(* Logix 5000 project; controller STAT 1756-L72 rev 20.12; software revision 20.04; part 2 of 34 *)
(* tags used below, declared in another part *)
   N7 : DINT[255];
   p15 : BOOL;
   P16 : BOOL;
   P17 : BOOL;
   P18 : BOOL;
   P23 : BOOL;
   P24 : BOOL;
   P3 : BOOL;
   P4 : BOOL;
   pd3 : BOOL;
   pd4 : BOOL;
   pd5 : BOOL;
   pd6 : BOOL;
   PD7 : BOOL;
   PD8 : BOOL;
   PM1 : BOOL;
   PM2 : BOOL;
   PM3 : BOOL;
   PM4 : BOOL;
   Q2 : REAL;
   Q3 : REAL;
   Q4 : REAL;
   real : REAL;
   S : INT[164];
   S1 : BOOL;
   Seconde : BOOL;

ADD_ON_INSTRUCTION integrat   (* revision 1.0 *)
VAR_INPUT
   rate : DINT; {required}
END_VAR
VAR_OUTPUT
   oai : DINT; {access Read Only, required}
END_VAR
VAR_INPUT
   AI : DINT; {required}
END_VAR
VAR
   memo : REAL; {access None}
   memo1 : REAL; {access None}
   rate1 : DINT; {access None}
   memo2 : REAL; {access None}
END_VAR

ROUTINE Logic   (* ladder *)
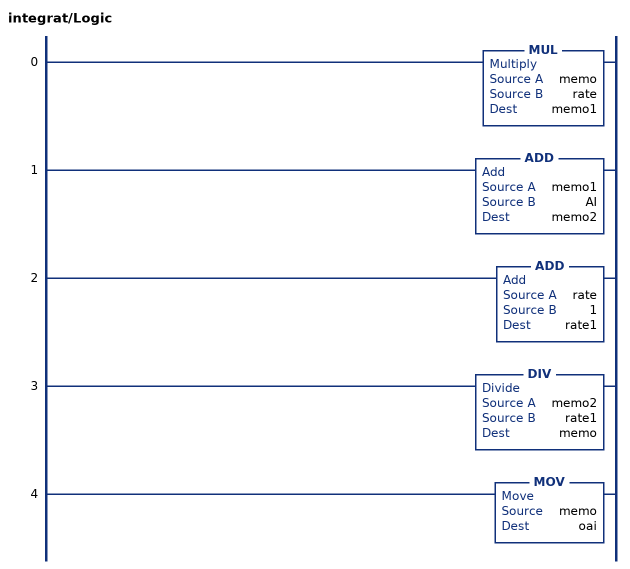
   0: MUL(memo,rate,memo1);
   1: ADD(memo1,AI,memo2);
   2: ADD(rate,1,rate1);
   3: DIV(memo2,rate1,memo);
   4: MOV(memo,oai);
END_ROUTINE
END_ADD_ON_INSTRUCTION

ADD_ON_INSTRUCTION SCP   (* revision 1.2, vendor Rockwell Automation *)
VAR_INPUT
   Input : REAL; {required}
   Input_Min : REAL; {required}
   Input_Max : REAL; {required}
   Scaled_Min : REAL; {required}
   Scaled_Max : REAL; {required}
END_VAR
VAR_OUTPUT
   Output : REAL; {access Read Only, required}
END_VAR
VAR
   Rate : REAL;
END_VAR

ROUTINE Logic   (* ladder *)
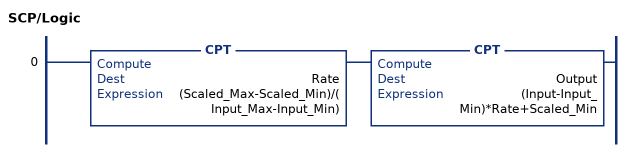
   0: CPT(Rate,(Scaled_Max-Scaled_Min)/(Input_Max-Input_Min))CPT(Output,(Input-Input_Min)*Rate+Scaled_Min);
END_ROUTINE
END_ADD_ON_INSTRUCTION

VAR_GLOBAL   (* controller tags *)
   ai_flow_L1 : REAL := 236.55;
   ai_flow_L2 : REAL := 242.7;
   ai_flow_L3 : REAL := 242.85;
   apport_soude_ibt_occupe : BOOL;
   aux2_P1 : BOOL := 1;
   AUX2_P2 : BOOL := 1;
   AUX_COND_KOELTOREN : REAL := 3777.7964;
   AUX_LVL_KOEL : DINT := 857;
   aux_P1_ETANG : BOOL := 1;
   AUX_P1P2 : BOOL;
   AUX_P2 : BOOL := 1;
   AUX_P5_RINC : BOOL;
   av310 : BOOL := 1;
   av320 : BOOL := 1;
   av330 : BOOL := 1;
   averflowput1 : DINT := -30;
   averflowput2 : DINT := -24;
   averK1 : DINT := 206;
   averK2 : DINT := 230;
   averL1 : DINT := 261;
   averL2 : DINT := 162;
   averL3 : DINT := 242;
   averlpmpput2 : DINT;
   averpmpput1 : DINT;
   averQ1 : DINT := 170;
   averQ2 : DINT := 131;
   B10 : DINT[20] := ([0] := 2#0000_0000_0000_0000_0010_1100_0100_0000, [1] := 2#0000_0000_0000_0000_0000_0000_0000_0101);
        [1].0   // b10:1/0
        [1].1   // b10:1/1
   B14 : DINT[30] := ([1] := 2#0000_0000_0000_0000_0000_0000_0000_1000, [2] := 2#0000_0000_0000_0000_0000_0000_0000_0010, [4] := 2#0000_0000_0000_0000_0010_0000_0000_0101, [5] := 2#0000_0000_0000_0000_0000_0100_1000_0011, [7] := 2#0000_0000_0000_0000_0000_0000_0000_0001, [11] := 2#0000_0000_0000_0000_0000_1000_0000_0001, [15] := 2#0000_0000_0000_0000_0000_0000_0000_0011, [16] := 2#0000_0000_0000_0000_0000_0000_0010_0000, [18] := 2#0000_0000_0000_0000_0000_0000_0000_0100, [19] := 2#0000_0000_0000_0000_0000_0000_0000_0101, [21] := 2#0000_0000_0000_0000_0000_0000_0001_0000, [23] := 2#0000_0000_0000_0000_0000_0000_1000_0000);
        [0].10   // Fout cls 2 noodstop gedrukt
        [0].11   // Fout cls 3 noodstop gedrukt
        [0].12   // Fout cls 4 noodstop gedrukt
        [0].13   // Fout stormbekken noodstop gedrukt
        [0].14   // Fout stormbekken noodstop relais is niet ok
        [1].0   // Fout cls 2 noodstop relais niet ok
        [1].1   // Fout cls 3 noodstop relais niet ok
        [1].2   // Fout cls 4 noodstop relais niet ok
        [1].3   // Fout cls 5 noodstop relais niet ok
        [1].4   // Fout eurowater noodstop relais niet ok
        [1].5   // Fout IBT A noodstop relais niet ok
        [1].6   // Fout IBT B noodstop relais niet ok
        [1].7   // Fout IBT C noodstop relais niet ok
        [1].10   // fout visu LACK DETECTIE NAOH
        [1].11   // fout visu LACK DETECTIE H2SO4
        [1].12   // Fout 24vdc algemeen
        [1].13   // Fout 24vdc ingangen
        [1].14   // Fout 24vdc instrument
        [1].15   // Fout 24vdc uitgangen
        [2].0   // Fout geen 220 V aan bedieningskast lijn 1 2 3 4
        [2].1   // FC NIVEAU CUVE AZ
        [2].2   // Fout geen 220 V aan stormbekken nuts
        [2].3   // Fout geen 220 V aan stormbekken stuurspanning
        [2].4   // Fout geen 24 V aan stormbekken stuurspanning
        [2].5   // Fout geen 220 V algemeen
        [2].6   // Fout geen voedingspanning lijn 1 cl2
        [2].7   // Fout geen voedingspanning lijn 2 cl3
        [2].8   // Fout geen voedingspanning lijn 3 cl4
        [2].9   // Fout geen voedingspanning lijn 4 cl5
        [2].10   // Fout geen voedingspanning eurow cl6
        [2].11   // Fout geen voedingspanning ibt a
        [2].12   // Fout geen voedingspanning ibt b
        [2].13   // Fout geen voedingspanning ibt c
        [2].14   // Fout geen voedingsspanning instrumenten
        [2].15   // fout voeding 24 v dc niet ok
        [3].0   // ???
        [3].1   // ???
        [3].2   // ???
        [4].0   // Fout niveau lus 5
        [4].1   // Fout niveau lus 6
        [4].2   // Fout niveau vlotter A3
        [4].3   // Fout niveau lus 7
        [4].11   // defaut VANNE ALIBERT
        [4].12   // defaut vanne pmp puits 2
        [4].13   // defaut vanne pmp puits 3
        [9].0   // resetmerker die in visualisatie hoog wordt gezet
        [10].0   // pomp 1 thermische storing
        [10].2   // pomp 2 thermische storing
        [10].4   // p3 fout thermische storing
        [10].6   // fout geen spanning freqreg pd1
        [10].7   // fout nivea van cuve 3 voor het spoelen van ontijzer
        [10].8   // fout nivea van lus4 voor het spoelen van ontijzer
        [10].9   // fout geen spanning freqreg pd2
        [10].10   // fout thermische storing motor pd2
        [10].11   // fout vlotter lal 1
        [10].12   // fout promag 33 storing
        [10].14   // FOUT_CA1
        [10].15   // S1 thermische storing
        [11].0   // p3 thermische storing
        [11].1   // p3 storing niet op tijd in driehoek
        [11].2   // p4 thermische storing
        [11].3   // EV3_TIJDBEV
        [11].4   // p5 thermische storing
        [11].5   // p6 thermische storing
        [11].6   // FOUT_EV6_TIJDBEV
        [11].7   // FOUT_EV7_TIJDBEV
        [11].8   // FOUT_NIV_DOUBLE_MAX
        [11].9   // FOUT_NIV_DOUBLE_MIN
        [11].10   // p25 fout geen spanning op freqreg
        [11].11   // P25_FOUT_KLEP_EV2
        [11].12   // p25 fout frequentieregelaar storing
        [12].0   // p11 fout thermische storing
        [12].1   // p12 fout thermische storing
        [12].2   // fout conductiviteit 3
        [12].3   // FOUT_COND3_NIET_OK
        [13].0   // p13 fout thermische storing
        [13].1   // p14 fout thermische storing
        [13].2   // FOUT_CON4
        [13].3   // FOUT_COND4_NIET_OK
        [13].10   // FOUT_COND1_NIET_OK
        [13].11   // FOUT_COND1_MAX
        [13].13   // FOUT_COND2_NIET_OK
        [13].14   // FOUT_COND2_MAX
        [14].0   // p15 fout thermische storing
        [14].1   // p16 fout thermische storing
        [14].2   // FOUT_CON5
        [14].3   // FOUT_COND5_NIET_OK
        [15].0   // p17 fout thermische storing
        [15].1   // p18 fout thermische storing
        [15].2   // FOUT_CON6
        [15].3   // FOUT_COND6_NIET_OK
        [16].0   // Fout maximum niveau lus 1
        [16].1   // Fout minimum niveau lus 1
        [16].3   // conductivit?trop grande trop longtemps arret P1.1 & P1.2
        [16].5   // Fout debietmeter Q2
        [16].6   // Fout debietmeter Q3
        [16].7   // FOUT_DEBIETM_Q4
        [17].0   // Fout thermische storing pro1
        [17].1   // STORING_OSM1_COND niet ok na tijd
        [17].2   // Fout thermische storing pro2
        [17].3   // STORING_OSM2_COND niet ok na tijd
        [17].4   // Fout thermische storing pro3
        [17].5   // STORING_OSM3_COND niet ok na tijd
        [17].6   // Fout thermische storing p7
        [17].8   // Fout thermische storing p8
        [17].10   // Fout thermische storing p9
        [17].11   // ???
        [17].12   // FOUT_THST_P21_AZ
        [17].14   // Fout thermische storing p22 kuip az
        [18].0   // Fout thermische storing p21 reiniging
        [18].1   // Fout thermische storing s1 ventilator
        [18].2   // Fout thermische storing s1
        [18].10   // FOUT_OSM1_DRUK
        [18].11   // FOUT_OSM2_DRUK
        [18].12   // FOUT_OSM3_DRUK
        [19].0   // Fout thermische storing p23 kelder
        [19].2   // Fout thermische storing p24 kelder
        [19].6   // Fout thermische storing AG1 mixer
        [19].8   // Fout thermische storing AG2 mixer
        [19].10   // Fout thermische storing AG3 mixer
        [19].11   // OPVULLEN_TANK_1
        [20].0   // Fout thermische storing pd3 dos ac
        [20].2   // Fout thermische storing pd4 dos ac
        [20].4   // Fout thermische storing pd5 dos ac
        [20].6   // Fout thermische storing pd6 dos ac
        [20].10   // FOUT_PH11_12_STORING
        [20].11   // FOUT_PH11_ZUUR
        [20].12   // FOUT_PH11_BAZE
        [20].13   // FOUT_PH11_12_ABS_MAX
        [20].14   // FOUT_PH_LAAG
        [20].15   // FOUT_PH_HOOG
        [21].0   // FOUT_THST_PD7
        [21].2   // FOUT_THST_PD8
        [21].4   // FOUT_THST_P19A
        [21].5   // FOUT_THST_P19B
        [21].6   // FOUT_THST_PM1
        [21].7   // FOUT_THST_PM2
        [21].8   // FOUT_THST_PM3
        [21].9   // FOUT_THST_PM4
        [21].10   // FOUT_PH11_2_STORING
        [21].11   // PM1_MAX_DRUK
        [21].12   // PM1_GEEN_DEBIET
        [21].13   // PM2_MAX_DRUK
        [21].14   // PM2_GEEN_DEBIET
        [22].4   // FOUT_NIV_MAX_LAH6
        [22].5   // FOUT_NIV_MIN_LAH6
        [22].8   // PM3_MAX_DRUK
        [22].9   // PM3_GEEN_DEBIET
        [22].10   // PM4_MAX_DRUK
        [22].11   // PM4_GEEN_DEBIET
        [22].13   // FOUT_NIV_LAAG_LUS2
        [22].14   // FOUT_NIV_LUS2
        [23].0   // FOUT_NIV_LAAG_LUS3
        [23].1   // FOUT_NIV_LUS3
        [23].3   // FOUT_NIV_MAX_CUVE3
        [23].4   // FOUT_NIV_MIN_CUVE3
        [23].6   // FOUT_NIV_MAX_LU4
        [23].7   // FOUT_NIV_MIN_LUS4
   B15 : DINT[30] := ([7] := 2#0000_0000_0000_0000_0000_0000_0000_0011, [11] := 2#0000_0000_0000_0000_0000_1000_0000_0001, [15] := 2#0000_0000_0000_0000_0000_0000_0000_0011, [16] := 2#0000_0000_0000_0000_0000_0000_0010_0000, [18] := 2#0000_0000_0000_0000_0000_0000_0000_0100, [19] := 2#0000_0000_0000_0000_0000_0000_0000_0101, [21] := 2#0000_0000_0000_0000_0000_0000_0001_0000, [23] := 2#0000_0000_0000_0000_0000_0000_1000_0000);
   B16 : DINT[30] := ([1] := 2#0000_0000_0000_0000_0000_0000_0000_0011, [9] := 2#0000_0000_0000_0000_0000_0000_0000_1000, [10] := 2#0000_0000_0000_0000_0011_1001_0000_0000, [11] := 2#0000_0000_0000_0000_0100_0100_0000_0001, [14] := 2#0000_0000_0000_0000_0000_0000_0001_0100);
        [10].0   // flank omschakelen van aandrijving na dag
        [10].1   // flank bij omschakeling na dag draaien
        [10].2   // flank debietmeting Q1
        [10].3   // flank omschakelen van aandrijving na dag bij hoog timer
        [10].4   // flank omschakelen van aandrijving na dag bij laag timer
        [10].5   // flank q1 debiet ontijzering 2
        [10].6   // flank q1 tfb1.2 in bedrijf nemen
        [10].7   // flank q1 tfb1.1 in bedrijf nemen
        [10].8   // flank debiet promag 33
        [10].9   // Flank reinigen ontijzer 1
        [10].11   // FLANK_DEBIET_Q2
        [10].14   // Hand osmose 3 ster driehoek
        [11].0   // Hulp merker flank als er geen osmose motoren draaien
        [11].1   // Flank als er geen osmose motoren draaien
        [11].11   // one shot
   B17 : DINT[30] := ([1] := 2#0000_0000_0000_0000_0000_0000_0000_0100, [3] := 2#0000_0000_0000_0000_0001_0000_0000_0000, [10] := 2#0000_0000_0000_0000_0000_0011_0000_0111, [11] := 2#0000_0000_0000_0000_1010_0000_1100_0001, [12] := 2#0000_0000_0000_0000_0100_0100_0000_1000, [13] := 2#0000_0000_0000_0000_0000_0000_0100_0000, [15] := 2#0000_0000_0000_0000_0000_0000_0000_0001, [16] := 2#0000_0000_0000_0000_0000_0000_0000_1111, [17] := 2#0000_0000_0000_0000_0000_0000_1100_0001);
        [1].1   // bp supervis passage etang<>puits
        [1].2   // pmp etang
        [1].3   // pmp puits
        [1].4   // ons
        [1].5   // demande changement pmp etang <> puits
        [1].6   // choix pompe puits
        [10].0   // keuzebit pomp 1 of pomp 2 om beurt draaien
        [10].1   // ontijzering kan draaien en is ok
        [10].2   // verzachter is ok er kan water door
        [10].3   // hoog is keuze ontijzering 1
        [10].4   // hoog is keuze verzachter 1
        [10].5   // reinig ontijzer 1
        [10].6   // reinig ontijzer 2
        [10].7   // backwach 1 in bedrijf nemen
        [10].8   // backwach 2 in bedrijf nemen
        [10].11   // Automaat osmose 2 ster driehoek
        [10].12   // bp bypass osmose
        [10].14   // Automaat osmose 3 ster driehoek
        [10].15   // choix marche 2pmp
        [11].3   // keuze pd1 of pd2
        [11].4   // eau pretraite
        [11].5   // LSH_HOOG_LUS1
        [11].6   // LSL1_LAAG_LUS1
        [11].7   // LAL2_LAAG_LUS1
        [11].8   // niveau bas vijver pour P1
        [11].10   // keuze pomp 3 of pomp 4
        [11].11   // keuze pomp 5 of pomp 6
        [11].13   // keuze pomp 11 of pomp 12
        [11].15   // keuze pomp 13 of pomp 14
        [12].1   // keuze pomp 15 of pomp 16
        [12].3   // keuze pomp 17 of pomp 18
        [12].10   // Pompen p11 tot p18 mogen pompen naar cuve nr4
        [12].11   // conductieviteit 3 is ok pompen p11 of p12 mogen draaien
        [12].12   // conductieviteit 4 is ok pompen p13 of p14 mogen draaien
        [12].13   // conductieviteit 5 is ok pompen p15 of p16 mogen draaien
        [12].14   // conductieviteit 6 is ok pompen p17 of p18 mogen draaien
        [13].0   // ?
        [13].6   // osmose 1 wordt vrijgegeven om te draaien
        [13].7   // osmose 2 wordt vrijgegeven om te draaien
        [13].8   // osmose 3 wordt vrijgegeven om te draaien
        [13].9   // Aanvraag tot reinigen osmose 1
        [13].10   // Aanvraag tot reinigen osmose 2
        [13].11   // Aanvraag tot reinigen osmose 3
        [13].12   // ??
        [13].13   // ?
        [13].14   // Start reinigen duble M
        [14].0   // Aanvraag tot reinigen onteizering 1 van osmose
        [14].1   // Aanvraag tot reinigen onteizering 2 van osmose
        [14].2   // Regenereer ontharder recup water 1
        [14].3   // Regenereer ontharder recup water 2
        [14].7   // osmose reiniging met zuur is gekozen en bezig
        [14].8   // osmose reiniging met base is gekozen en bezig
        [14].9   // osmose reiniging met lang is gekozen en bezig
        [15].0   // keuzebit pomp 21 of pomp 22
        [15].12   // keuzebit pomp 23 of pomp 24
        [16].0   // NIV_LUS_4_ONDER1
        [16].1   // NIV_LUS_4_ONDER2
        [16].2   // NIV_LUS_4_BOVEN3
        [16].3   // NIV_LUS_4_BOVEN4
        [17].0   // keuzebit pomp pd3 pd4
        [17].1   // zuur toevoegen pd3 of pd4
        [17].2   // keuzebit pomp pd5 pd6
        [17].4   // KEUZEBIT_P19_P20
        [17].5   // KEUZEBIT_PD7_PD8
        [17].6   // P11_TOT_P18_DRAAIEN
        [17].7   // P11_TOT_P18_T27_80
        [18].0   // supervision start].stop PM1
        [18].1   // supervision start].stop PM2
        [18].4   // supervision start].stop PM3
        [18].5   // supervision start].stop PM4
   B25 : DINT[30] := ([0] := 2#0000_0000_0000_0000_0000_0000_0000_0010, [1] := 2#0000_0000_0000_0000_0000_0000_0000_0010);
        [0].0   // Pomp p11 p12 aan auto syclus
        [0].1   // Keuzebit lijn 1 pomp 11 of pomp 12
        [0].4   // Pomp p13 p14 aan auto syclus
        [0].5   // Keuzebit lijn 1 pomp 13 of pomp 14
        [0].6   // ?
        [0].8   // POMP_P15_P16_AANN
        [0].9   // Keuzebit lijn 1 pomp 15 of pomp 16
        [0].12   // POMP_P17_P18_AAN
        [0].13   // KEUZEBIT_P17_OF_P18
        [1].0   // Osmose pompen draaien 1
        [1].1   // Twee pompen aan bij voeding osmose 123
        [1].6   // Osmose pompen draaien 2
        [1].12   // Osmose pompen draaien 3
   B3 : DINT[256] := ([0] := 2#0000_0000_0000_0000_0100_0000_0000_0110, [1] := 2#0000_0000_0000_0000_0010_0110_1100_1001, [2] := 2#0000_0000_0000_0000_0000_0000_0000_0001, [3] := 2#0000_0000_0000_0000_0000_0000_0000_0010, [4] := 2#0000_0000_0000_0000_0000_0000_0000_0111, [5] := 2#0000_0000_0000_0000_0000_0000_0000_0001, [6] := 2#0000_0000_0000_0000_0000_0000_0000_0110, [7] := 2#0000_0000_0000_0000_0000_0000_1010_0110, [8] := 2#0000_0000_0000_0000_0000_0000_0001_0010, [9] := 2#0000_0000_0000_0000_0000_0000_0001_0010, [10] := 2#0000_0000_0000_0000_0111_1000_0000_0111, [12] := 2#0000_0000_0000_0000_0000_0010_0111_1001, [15] := 2#0000_0000_0000_0000_1000_0100_1000_0111, [17] := 2#0000_0000_0000_0000_0001_0100_0001_0001, [18] := 2#0000_0000_0000_0000_0000_0000_1000_1000, [19] := 2#0000_0000_0000_0000_0000_0010_0000_0010, [20] := 2#0000_0000_0000_0000_0000_0001_0111_0010, [21] := 2#0000_0000_0000_0000_0000_0000_0000_1110, [22] := 2#0000_0000_0000_0000_0000_0000_0100_0011, [23] := 2#0000_0000_0000_0000_0000_0000_0100_0000, [24] := 2#0000_0000_0000_0000_0000_0000_1111_0000, [26] := 2#0000_0000_0000_0000_0000_0000_0000_0100, [28] := 2#0000_0000_0000_0000_0000_0000_0000_0100, [29] := 2#0000_0000_0000_0000_0000_0000_0011_1111, [30] := 2#0000_0000_0000_0000_0000_0000_0100_0000, [31] := 2#0000_0000_0000_0000_0000_1000_0000_0000, [34] := 2#0000_0000_0000_0000_0000_0000_0000_0100, [41] := 2#0000_0000_0000_0000_0000_0000_0000_1000, [42] := 2#0000_0000_0000_0000_0000_0000_0000_0010, [44] := 2#0000_0000_0000_0000_0010_0000_0000_0101, [45] := 2#0000_0000_0000_0000_0000_0100_1000_0011, [47] := 2#0000_0000_0000_0000_0000_0000_0000_0001, [51] := 2#0000_0000_0000_0000_0000_1000_0000_0001, [55] := 2#0000_0000_0000_0000_0000_0000_0000_0011, [56] := 2#0000_0000_0000_0000_0000_0000_0010_0000, [58] := 2#0000_0000_0000_0000_0000_0000_0000_0100, [59] := 2#0000_0000_0000_0000_0000_0000_0000_0101, [61] := 2#0000_0000_0000_0000_0000_0000_0001_0000, [63] := 2#0000_0000_0000_0000_0000_0000_1000_0000, [65] := 2#0000_0000_0000_0000_0001_0000_0000_0100, [66] := 2#0000_0000_0000_0000_0000_0011_0000_0001, [67] := 2#0000_0000_0000_0000_1010_0000_0000_0000, [69] := 2#0000_0000_0000_0000_0000_0000_0100_0000, [70] := 2#0000_0000_0000_0000_0011_1111_1100_0001, [73] := 2#0000_0000_0000_0000_0010_1100_0100_0000, [74] := 2#0000_0000_0000_0000_0000_0000_0000_0101, [80] := 2#0000_0000_0000_0000_0000_0000_0000_0001, [81] := 2#0000_0000_0000_0000_0000_0000_0000_0001, [82] := 2#0000_0000_0000_0000_0000_0000_0000_0001, [83] := 2#0000_0000_0000_0000_0000_0000_0010_0000, [84] := 2#0000_0000_0000_0000_0000_0000_0000_0001, [85] := 2#0000_0000_0000_0000_0000_0000_0100_0000, [86] := 2#0000_0000_0000_0000_0000_0000_0000_0001, [87] := 2#0000_0000_0000_0000_0000_0000_0000_0100, [88] := 2#0000_0000_0000_0000_0000_0000_0000_0001, [89] := 2#0000_0000_0000_0000_0000_0000_0000_0001, [90] := 2#0000_0000_0000_0000_0000_0000_0000_0001, [91] := 2#0000_0000_0000_0000_0000_0000_0000_0001, [92] := 2#0000_0000_0000_0000_0000_0000_0000_0001, [93] := 2#0000_0000_0000_0000_0000_0000_0000_0011,
        [94] := 2#1111_1111_1111_1111_1100_1000_1001_1000, [95] := 2#0000_0000_0000_0000_0111_0100_1101_0000, [96] := 2#0000_0000_0000_0000_0000_0000_0000_1000, [97] := 2#0000_0000_0000_0000_0001_0000_0000_0000, [98] := 2#1111_1111_1111_1111_1000_0000_0000_0000, [99] := 2#0000_0000_0000_0000_0011_0000_0010_0010, [101] := 2#0000_0000_0000_0000_0000_0000_1000_0000, [102] := 2#0000_0000_0000_0000_0000_0000_0001_0100, [103] := 2#1111_1111_1111_1111_1111_1111_0100_0000, [104] := 2#0000_0000_0000_0000_0000_0000_0111_1111, [105] := 2#1111_1111_1111_1111_1000_1000_1011_1111, [106] := 2#0000_0000_0000_0000_0101_1101_1000_0110, [107] := 2#1111_1111_1111_1111_1000_1011_1000_0111, [108] := 2#0000_0000_0000_0000_0010_1000_1000_1000, [109] := 2#1111_1111_1111_1111_1000_0101_0111_1000, [110] := 2#1111_1111_1111_1111_1010_1110_1011_1111, [111] := 2#1111_1111_1111_1111_1111_1110_0011_1111, [112] := 2#0000_0000_0000_0000_0110_0111_0111_1111, [113] := 2#1111_1111_1111_1111_1001_1100_0001_0000, [114] := 2#0000_0000_0000_0000_0010_0011_0110_0000, [115] := 2#1111_1111_1111_1111_1100_0000_0111_1110, [116] := 2#0000_0000_0000_0000_0000_0000_0000_0110, [117] := 2#1111_1111_1111_1111_1010_1010_0000_0000, [120] := 2#1010_1010_1010_1010_0000_0000_0000_0110, [121] := 2#0000_0000_0000_0000_0000_0000_0000_0110, [122] := 2#0000_0000_0000_0110_1010_1010_1010_1010, [123] := 2#0000_0000_0000_0000_1010_1010_1010_1010, [124] := 2#0001_0000_0000_0000_0000_0000_0000_0000);
        [0].1   // ???
        [0].4   // b3:0/4
        [0].5   // FLOW TOO LOW Q1
        [0].6   // def flow Q1
        [0].7   // def flow Q2
        [0].8   // FLOW TOO LOW Q2
        [0].10   // aux klaxon NAOH
        [0].11   // aux klaxon H2SO4
        [0].12   // aux klaxon ZOUT
        [0].13   // ons
        [0].14   // ons
        [0].15   // ons
        [1].4   // ouverture EV7 + P6
        [1].8   // re-init flex I].O
        [7].0   // START P23 by ventury
        [7].1   // ??
        [7].2   // ??
        [7].3   // DEMARRE PMP L4 niveau puisard
        [7].4   // demarrage niveau pmp 1 puisard ligne 4
        [7].5   // demarrage niveau pmp 2 puisard ligne 4
        [7].6   // ??
        [7].7   // one shot
        [8].0   // osmose 2 en cours
        [8].1   // osmose 1 en cours
        [8].2   // osmose 3 en cours
        [8].4   // DEMANDE DEMARRAGE AU MOINS 1 POMPE
        [8].5   // DEMANDE DEMARRAGE AU MOINS 2 POMPES
        [8].6   // DEMANDE DEMARRAGE AU MOINS 3 POMPES
        [9].1   // Smeermerker
        [9].2   // Smeermerker 2
        [9].3   // Ingang therm st
        [9].4   // mot uitg aan
        [9].5   // SMEERM5
        [9].6   // SMEERM6
        [9].7   // SMEERM7
        [9].8   // SMEERM8
        [9].9   // SMEERM9
        [9].10   // SMEERM10
        [9].11   // SMEERM11
        [9].12   // SMEERM12
        [9].13   // SMEERM13
        [9].14   // SMEERM14
        [9].15   // SMEERM15
        [10].0   // de ftv acquit
        [10].1   // flank iedere 10 sec
        [10].2   // FLANK_IEDERE_MIN
        [10].9   // Algemeen sturing in en noodstoppen ok
        [10].10   // sturing is in via visual
        [10].11   // verzachter 1 autom aan
        [10].12   // verzacherter 2 automaat aan
        [10].13   // ontijzer 1 aan
        [10].14   // ontijzer 2 aan
        [11].11   // start backwach ontharder 1
        [11].12   // start backwach ontharder 2
        [11].13   // ontijzer1 start backwach
        [11].14   // ontijzer2 start backwach
        [12].0   // P3 en P4 aan aan via visual
        [12].1   // pomp p5 en p6 aan
        [12].5   // p25 aan via visual
        [12].7   // p11 tot p18 aan via visual
        [13].0   // pro 1 tot 3 aan via visualisatie
        [14].0   // pomp p7 8 9 aan via visualisatie
        [14].1   // pomp p21 en 22 aan via visual
        [14].3   // pomp p21 reinigingsopmp aan
        [14].4   // Vent s1 reinigingsvent
        [14].5   // VISUAL_TANK_1_VUL
        [14].6   // VISUAL_TANK_2_VUL
        [14].10   // pomp p23 24 aan via visual
        [14].11   // AG1 2 3 aan via visual
        [14].14   // PD3 en PD4 aan via visual
        [15].0   // Automaat duble M aan
        [15].1   // Automaat verzachter recup water 1
        [15].2   // AUTOM_VERZREC2
        [15].3   // Forceer backwach duble M
        [15].4   // forceer regeneren verzachter recupwater 1
        [15].5   // FORCE_REGEN_VERZREC2
        [15].7   // de superv auto RO1
        [15].8   // MAN].AUTO depuis sup OSMOSE 2
        [15].9   // de superv auto RO3
        [15].10   // Automaat osmose 1 via visual
        [15].11   // Automaat osmose 2 via visual
        [15].12   // Automaat osmose 3 via visual
        [15].14   // de supervision by pass osmose
        [15].15   // AUTO_NEUTRAL
        [16].0   // Aanvraag reiniging via visual ro1 zuur
        [16].1   // Aanvraag reiniging via visual ro1 baze
        [16].2   // Aanvraag reiniging via visual ro1 lang
        [16].3   // Aanvraag reiniging via visual ro2 zuur
        [16].4   // Aanvraag reiniging via visual ro2 baze
        [16].5   // Aanvraag reiniging via visual ro2 lang
        [16].6   // Aanvraag reiniging via visual ro3 zuur
        [16].7   // Aanvraag reiniging via visual ro3 baze
        [16].8   // Aanvraag reiniging via visual ro3 lang
        [17].1   // ons P7 arret
        [17].3   // ons P8 arret
        [17].5   // ons P9 arret
        [17].9   // FL_STOP_RO1
        [17].11   // FL_STOP_RO2
        [17].13   // FL_STOP_RO3
        [18].1   // PRO1_LAATST_GESTOPT
        [18].2   // PRO2_LAATST_GESTOPT
        [18].3   // PRO3_LAATST_GESTOPT
        [18].7   // P7 est la derniere pompe arrete
        [18].8   // P8 est la derniere pompe arrete
        [18].9   // P9 est la derniere pompe arrete
        [19].1   // PRO1_VOORLA_GEST
        [19].2   // PRO2_VOORLA_GEST
        [19].3   // PRO3_VOORLA_GEST
        [19].7   // P7 est l'avant derniere pompe arrete
        [19].8   // P8 est l'avant derniere pompe arrete
        [19].9   // P9 est l'avant derniere pompe arrete
        [20].1   // une pompe P7,8 ou a enclench?,,,0,,,0,
        [20].2   // 2 pompe P7,8 ou 9 a enclench?,,,0,,,0,
        [20].3   // 3 pompe P7,8 ou 9 a enclench?,,,0,,,0,
        [20].4   // PRO1_DRAAI
        [20].5   // PRO2_DRAAI
        [20].6   // PRO3_DRAAI
        [20].7   // P7 doit tourner
        [20].8   // P8 doit tourner
        [20].9   // P9 doit tourner
        [21].1   // 1 pompe osmose ?demarrer
        [21].2   // 2 pompe osmose ?demarrer
        [21].3   // 3 pompe osmose ?demarrer
        [22].6   // ons
        [22].7   // ons stfa1 ev1
        [22].8   // ons
        [22].9   // ons stfa1 ev2
        [23].0   // demarrage PMP 21 pour nettoyage osmose
        [23].1   // auxiliaire demarrage PMP 21 pour nettoyage osmose
        [23].2   // auxiliaire demarrage PMP 21 pour nettoyage osmose
        [23].3   // marche manu PMP 21
        [23].4   // autorisation marche auto PMP 21
        [23].5   // demande marche auto PMP 21
        [23].7   // auxiliaire marche PMP 7 ?9
        [23].8   // ??
        [24].0   // ons
        [24].1   // ONS
        [24].2   // ONS
        [24].3   // ONS
        [24].4   // conditions PM1
        [24].5   // CONDITIONS PM2
        [24].6   // CONDITIONS PM3
        [24].7   // CONDITIONS PM4
        [24].8   // start].stop PM1
        [24].9   // start].stop PM2
        [24].10   // start].stop PM3
        [24].11   // start].stop PM4
        [26].0   // ARRET 1 pmp pm7 ?9
        [27].0   // demande marche pmp puits
        [28].0   // ons
        [28].1   // aux ons pmp 1
        [28].2   // ons
        [28].3   // aux ons pmp 2
        [28].4   // marche pmp 2
        [29].0   // test p1 l4
        [29].1   // test p2 l4
        [29].2   // test p23
        [29].3   // test p24
        [29].4   // test p19
        [29].5   // test p20
        [30].2   // changement de journe
        [30].9   // ons].seconde clock plc
        [31].8   // 1 heure passe
        [31].9   // record log data
        [31].12   // ons
        [31].13   // ons
        [32].0   // AJOUT SOUDE
        [32].1   // AJOUT ACIDE
        [34].2   // stop RO2
        [70].0   // flank bij stoppen osmose 1
        [70].1   // flank bij stoppen osmose 1
        [70].2   // flank bij stoppen osmose 2
        [70].3   // flank bij stoppen osmose 2
        [70].4   // flank bij stoppen osmose 3
        [70].5   // flank bij stoppen osmose 3
   B9 : DINT[40] := ([9] := 2#0000_0000_0000_0000_0000_0000_0000_0001, [10] := 2#0000_0000_0000_0000_0000_0000_0000_0001, [11] := 2#0000_0000_0000_0000_0000_0000_0000_0001, [12] := 2#0000_0000_0000_0000_0000_0000_0000_0001, [13] := 2#0000_0000_0000_0000_0000_0000_0010_0000, [14] := 2#0000_0000_0000_0000_0000_0000_0000_0001, [15] := 2#0000_0000_0000_0000_0000_0000_0100_0000, [16] := 2#0000_0000_0000_0000_0000_0000_0000_0001, [17] := 2#0000_0000_0000_0000_0000_0000_0000_0100, [18] := 2#0000_0000_0000_0000_0000_0000_0000_0001, [19] := 2#0000_0000_0000_0000_0000_0000_0000_0001, [20] := 2#0000_0000_0000_0000_0000_0000_0000_0001, [21] := 2#0000_0000_0000_0000_0000_0000_0000_0001, [22] := 2#0000_0000_0000_0000_0000_0000_0000_0001, [30] := 2#0000_0000_0000_0000_0000_0000_0000_1000);
        [10].1   // b9:10/1
        [12].0   // Stap 1 regenereer kolom 1
        [12].1   // Stap 1 regenereer kolom 1 bedrijf kolom 2
        [12].2   // Stap 2 afsluiten kolom 1
        [12].3   // Stap 3 opspoelen backwach
        [12].4   // Stap 4 pekelaanzuigen
        [12].5   // Stap 5 Naspoeling
        [12].6   // Stap 6 Standbij positie kolom 1
        [13].0   // STAP_0_IN_WERK_VERZ2
        [13].1   // STAP_1_REG2_BEDR1
        [13].2   // STAP_2_REG2_BEDR1
        [13].3   // STAP_3_SPOEL_BACKWA2
        [13].4   // STAP_4_PEKELAANZUIG2
        [13].5   // STAP_5_NASPOELEN_2
        [13].6   // STAP_6_STANDBY_2
        [14].0   // regeneration dual media filter stepp 0 always on except
        [14].1   // STAP1_DUALM
        [14].2   // STAP2_DUALM
        [14].3   // STAP3_DUALM
        [14].4   // STAP4_DUALM
        [14].5   // STAP5_DUALM
        [14].6   // STAP6_DUALM
        [14].7   // STAP7_DUALM
        [14].8   // STAP8_DUALM
        [14].9   // STAP9_DUALM
        [15].0   // STAP_0_IN_WERK_VERRC
        [15].1   // STAP_1_START_STFA32
        [15].2   // STAP_2_SLUIT_STFA32
        [15].3   // STAP_3_BACKW_STFA3
        [15].4   // STAP_4_RUST_STFA3
        [15].5   // STAP_5_RINCE_STFA3
        [15].6   // STAP_6_STANDB_STFA3
        [15].7   // STAP_7_END_STFA3
        [16].0   // STAP_0_IN_WERK_32
        [16].1   // STAP_1_START_STFA31
        [16].2   // STAP_2_SLUIT_STFA31
        [16].3   // STAP_3_BACKW_STFA32
        [16].4   // STAP_4_RUST_STFA32
        [16].5   // STAP_5_RINCE_STFA32
        [16].6   // STAP_6_STANDB_STFA32
        [16].7   // STAP_7_END_STFA32
        [17]   // step osmose 1
        [17].1   // osmose 1 etape prewash
        [17].3   // osmose 1 etape 3 bakwash
        [18].1   // osmose 2 etape prewash
        [18].3   // osmose 2 etape 3 bakwash
        [19].1   // osmose 3 etape prewash
        [19].3   // osmose 3 etape 3 bakwash
        [20]   // step
        [20].0   // step 0
        [20].1   // step 1
        [22]   // mot step rincage osmose zuur & baze
        [23].14   // de ftv
   BITMW1 : BOOL;
   BITMW2 : BOOL;
   C5 : COUNTER[15] := ([0].PRE := 10, [0].CU := 1, [1].PRE := 10, [1].CU := 1, [2].PRE := 10, [2].CU := 1, [3].PRE := 10, [3].CU := 1, [4].PRE := 10, [4].CU := 1, [5].PRE := 10, [5].CU := 1, [6].PRE := 10, [6].CU := 1, [7].PRE := 10, [7].ACC := 4, [7].CU := 1, [8].PRE := 10, [8].CU := 1, [9].PRE := 10, [9].ACC := 4, [9].CU := 1, [10].PRE := 10, [10].CU := 1, [11].PRE := 10, [11].CU := 1, [12].PRE := 20, [12].CU := 1);
   CDRO1 : REAL := 14.923324;
   CDRO2 : REAL;
   CDRO3 : REAL := 200.0;
   comm : BOOL := 1;
   COND1_EAURECYCL : REAL := -1250.0953;
   COND2_OSMOS : DINT := -307;
   COND3 : REAL := 358.4;
   COND4 : REAL := 257.5;
   COND7 : REAL := -0.0030517578;
   cond_6 : REAL := -489.5747;
   CONV_MSG_L1 : MESSAGE;
        MessageParameters(ServiceCode := 16#004c, LocalElement := N7[65], ...)
   CONV_MSG_R_bassin : MESSAGE;
        MessageParameters(ServiceCode := 16#0fa2, LocalElement := N[228], ...)
   CONV_MSG_R_lancy : MESSAGE;
        MessageParameters(ServiceCode := 16#0fa2, LocalElement := N[65], ...)
   CONV_MSG_w_lancy : MESSAGE;   // N11:50 dans N7:50
        MessageParameters(ServiceCode := 16#0faa, LocalElement := N[227], ...)
   DateTime : DINT[7] := ([0] := 2016, [1] := 10, [2] := 20, [3] := 15, [4] := 8, [5] := 20, [6] := 152629);   // DINT array tag for retrieve wallclock time through GSV created during conversion
        [0]   // Year
        [1]   // Month
        [2]   // Day
        [3]   // Hour
        [4]   // Minute
        [5]   // Second
        [6]   // Microsecond
   def1bassin : DINT;
   def2bassin : DINT;
   def_fow_ecotec : BOOL;
   def_temp_iwts : BOOL;
   dmd_h2so4_ibt_ok : BOOL;
   dmd_soude_ibt_ok : BOOL;
   EAU_VILLE : BOOL;
   F8 : REAL[256] := ([0] := 86400.0, [1] := 8640.0, [2] := 77001.0, [3] := 310298.0, [4] := 3483771.0, [5] := 3484227.0, [6] := 801745.0, [7] := 834023.0, [8] := 621669.0, [9] := 310607.0, [10] := -25.0, [11] := -25.003815, [12] := -30.0, [13] := -35.00534, [14] := 49.0, [15] := -725.1137, [16] := 801739.0, [17] := -25.003815, [18] := 15.0, [19] := 496.5557, [20] := -725.11035, [21] := 5.0, [22] := 77.0, [23] := 73.0, [24] := 75.0, [25] := 77.0, [26] := 66.0, [27] := 72.0, [28] := 834014.0, [29] := 22.0, [30] := 2.0, [32] := 75.0, [33] := 65.0, [34] := 85.0, [35] := 801483.0, [36] := 12175211.0, [37] := 3393327.0, [42] := -3364194.0, [43] := 486083.0, [44] := 6236138.0, [45] := 0.013611111, [46] := 432544.34, [48] := 50.0, [49] := 621485.0, [50] := -25.003815, [51] := -400.06082, [52] := -25.003801, [54] := 818976.0, [55] := 684918.0, [56] := 373934.0, [57] := 149581.0, [60] := 841.0, [61] := 340.0784, [62] := 342.1696, [63] := 17107.648, [64] := 17450.648, [65] := 262969.0, [66] := 180861.0, [67] := 142970.0, [68] := 139156.0,
        [69] := 227936.0, [70] := 203522.0, [71] := 131625.0, [72] := 65800.0, [73] := 53300.0, [74] := -21025.0, [75] := -25230.0, [76] := 180675.81, [77] := 66991.336, [78] := 159950.5, [79] := 598.101, [80] := 180668.12, [81] := 66985.336, [82] := 66393.234, [83] := 594.8018, [84] := 180081.02, [85] := 1280.3794, [86] := 80.02371, [87] := 5874.036, [88] := 38.9009, [89] := 467.99988, [90] := 77.99998, [95] := -30.004578, [96] := 0.01824065, [97] := -30.0, [100] := 75.20038, [101] := 350.0, [102] := 340.0, [103] := 360.0, [110] := 801745.0, [111] := 834023.0, [112] := 621669.0, [113] := 310607.0, [114] := 180668.12, [115] := 66985.336);
        [5]   // total debiet zandfilter m?
        [6]   // flow Q1 TOT
        [7]   // Q2 tot
        [8]   // Q3 tot
        [9]   // total debiet osmose
        [10]   // debit put 2
        [11]   // debit put 1
        [12]   // debit put 3
        [13]   // ph venturi
        [14]   // debit venturi
        [15]   // conductivite venturi
        [16]   // memo Q1
        [17]   // tEMPERATURE venturi
        [18]   // flow Q1 en X min
        [19]   // niveau puisard l1,2,3
        [20]   // conductivite venturi
        [21]   // PARAM seuil mini flow Q1 en X min
        [28]   // MEMO TOT Q2
        [29]   // DELTA Q2 EN X MIN
        [30]   // PARAM seuil mini flow Q2 en X min
        [46]   // total eau passe venturi depi 3].10].2010
        [50]   // debit put 2
        [51]   // debit put 2
        [54]   // ontizer 1
        [55]   // ontizer 2
        [56]   // osmoze
        [57]   // debit verzacher
        [60]   // comptage des secondes
        [65]   // average level landeniaan L1 aux
        [66]   // average level kijtlaag k1 aux
        [67]   // average level Quartair Q1 aux
        [68]   // average level Landeniaan L2 aux
        [69]   // average level Krijtlaag K2 aux
        [70]   // average level landeniaan L3 aux
        [71]   // average level quartair Q2 aux
        [72]   // % run].heure pmp put 2 aux
        [73]   // % run].heure pmp put 3 aux
        [74]   // average flow pmp put 2 aux
        [75]   // average flow pmp put 3 aux
        [76]   // total d?it puits 2
        [77]   // total debit puit 1
        [80]   // tot put 2
        [81]   // tot put 1
        [85]   // aux LEVEL TANK RECUP L3
        [86]   // LEVEL TANK RECUP L3
        [89]   // f8:89
        [90]   // f8:89
        [100]   // variation de vitesse
   FL_STOP_RO : BOOL;
   FLW_CO1 : REAL := 44.998856;
   FLW_CO2 : REAL;
   FLW_CO3 : REAL := 0.030518044;
   FLW_EAU_VILLE : REAL;
   FLW_PO1 : REAL := 171.36646;
   FLW_PO2 : REAL;
   FLW_PO3 : REAL := 0.091554135;
   ForceStatus : INT := 3;   // INT tag to retrieve Force enabled value through GSV created during conversion
   FRANCK : BOOL;
   GEN_FOUT : BOOL;
   h2so4_ibt_finit : BOOL;
   hard : REAL := -25.001907;
   I1 : INT[32] := ([0] := 2#0000_1111_0100_0001, [1] := 2#1111_1111_0100_0000, [5] := 2#1000_0001_0000_0000, [8] := 2#0010_1010_1010_1010, [9] := 2#1000_1000_1011_1111, [10] := 2#0000_0111_1110_1101, [16] := 2#0001_1111_1010_1010, [17] := 2#0110_1111_1010_1010, [18] := 2#0011_1111_1010_1010, [19] := 2#0000_0000_0000_1111);
   I10 : INT[2] := ([0] := 2#1010_1010_1010_1010, [1] := 2#1010_1010_1010_1010);
   I10_000_Bit00 : ALIAS FOR I10[0].0;   // Drukknop start CL7 P 19A
   I10_000_Bit01 : ALIAS FOR I10[0].1;   // Drukknop stop CL7 P 19A
   I10_000_Bit02 : ALIAS FOR I10[0].2;   // Drukknop start CL7 P 19B
   I10_000_Bit03 : ALIAS FOR I10[0].3;   // Drukknop stop CL7 P 19B
   I10_000_Bit04 : ALIAS FOR I10[0].4;   // Drukknop start CL7 res
   I10_000_Bit05 : ALIAS FOR I10[0].5;   // Stop CL7 reserve
   I10_000_Bit06 : ALIAS FOR I10[0].6;   // Noodstop gedrukt CL7
   I10_000_Bit07 : ALIAS FOR I10[0].7;   // Hand Automaat CL8
   I10_000_Bit08 : ALIAS FOR I10[0].8;   // Drukknop start CL8 P 20
   I10_000_Bit09 : ALIAS FOR I10[0].9;   // Drukknop stop CL8 P 20
   I10_000_Bit10 : ALIAS FOR I10[0].10;   // Drukknop start CL8 PM1
   I10_000_Bit11 : ALIAS FOR I10[0].11;   // Drukknop stop CL8 PM1
   I10_000_Bit12 : ALIAS FOR I10[0].12;   // Drukknop start CL8 PM2
   I10_000_Bit13 : ALIAS FOR I10[0].13;   // Drukknop stop CL8 PM2
   I10_000_Bit14 : ALIAS FOR I10[0].14;   // Drukknop start CL8 PM3
   I10_000_Bit15 : ALIAS FOR I10[0].15;   // Drukknop stop CL8 PM3
   I10_001_Bit00 : ALIAS FOR I10[1].0;   // Drukknop start CL8 PM4
   I10_001_Bit01 : ALIAS FOR I10[1].1;   // Drukknop stop CL8 PM4
   I10_001_Bit02 : ALIAS FOR I10[1].2;   // Drukknop open EV 1
   I10_001_Bit03 : ALIAS FOR I10[1].3;   // Drukknop toe EV 1
   I10_001_Bit04 : ALIAS FOR I10[1].4;   // Drukknop start reserv CL8
   I10_001_Bit05 : ALIAS FOR I10[1].5;
   I10_001_Bit06 : ALIAS FOR I10[1].6;   // Noodstop gedrukt CL9
   I10_001_Bit07 : ALIAS FOR I10[1].7;   // Hand Automaat CL9
   I10_001_Bit08 : ALIAS FOR I10[1].8;   // Drukknop start P9 CL9
   I10_001_Bit09 : ALIAS FOR I10[1].9;   // Drukknop stop P7 CL9
   I10_001_Bit10 : ALIAS FOR I10[1].10;   // Drukknop start P8 CL9
   I10_001_Bit11 : ALIAS FOR I10[1].11;   // Drukknop stop P8 CL9
   I10_001_Bit12 : ALIAS FOR I10[1].12;   // Drukknop start P9 CL9
   I10_001_Bit13 : ALIAS FOR I10[1].13;   // Drukknop stop P9 CL9
   I10_001_Bit14 : ALIAS FOR I10[1].14;   // Drukknop start reserve CL9
   I10_001_Bit15 : ALIAS FOR I10[1].15;   // Drukknop stop reserve CL9
   I19 : INT[2] := ([0] := 2#1010_0111_1011_0001, [1] := 2#0000_0001_0101_0110);
   I19_000_Bit00 : ALIAS FOR I19[0].0;   // VANNE ALIBERT OUVERTE
   I19_000_Bit01 : ALIAS FOR I19[0].1;   // VANNE ALIBERT FERMEE
   I19_000_Bit02 : ALIAS FOR I19[0].2;   // vanne pmp puit 3 ouverte
   I19_000_Bit03 : ALIAS FOR I19[0].3;   // vanne pmp puit 3 fermee
   I19_000_Bit04 : ALIAS FOR I19[0].4;   // vanne pmp puit 2 ouverte
   I19_000_Bit05 : ALIAS FOR I19[0].5;   // vanne pmp puit 2 fermee
   I19_000_Bit06 : ALIAS FOR I19[0].6;
   I19_000_Bit07 : ALIAS FOR I19[0].7;   // LACK DETECTIE H2SO4
   I19_000_Bit08 : ALIAS FOR I19[0].8;   // LACK DETECTIE NAOH
   I19_000_Bit09 : ALIAS FOR I19[0].9;   // BP RESET KLAXON
   I19_000_Bit10 : ALIAS FOR I19[0].10;   // by pass vers osmose
   I19_000_Bit11 : ALIAS FOR I19[0].11;   // by pass vers osmose
   I19_000_Bit12 : ALIAS FOR I19[0].12;   // pulse puit put 1
   I19_000_Bit13 : ALIAS FOR I19[0].13;   // puit put 2
   I19_000_Bit14 : ALIAS FOR I19[0].14;   // vanne eau ville open
   I19_000_Bit15 : ALIAS FOR I19[0].15;   // vanne eau ville closed
   I19_001_Bit00 : ALIAS FOR I19[1].0;   // pulse eau de ville
   I19_001_Bit01 : ALIAS FOR I19[1].1;   // Thermische beveiligneing pomp p23 in kelderkuip
   I19_001_Bit02 : ALIAS FOR I19[1].2;
   I19_001_Bit03 : ALIAS FOR I19[1].3;   // Thermische beveiligneing pomp p24 in kelderkuip
   I19_001_Bit04 : ALIAS FOR I19[1].4;
   I19_001_Bit05 : ALIAS FOR I19[1].5;   // vanne acide de stock fermee
   I19_001_Bit06 : ALIAS FOR I19[1].6;   // vanne acide de stock ouverte
   I19_001_Bit07 : ALIAS FOR I19[1].7;   // vanne soude de stock ouverte
   I19_001_Bit08 : ALIAS FOR I19[1].8;   // vanne soude de stock fermée
   I19_001_Bit09 : ALIAS FOR I19[1].9;
   I19_001_Bit10 : ALIAS FOR I19[1].10;
   I19_001_Bit11 : ALIAS FOR I19[1].11;
   I19_001_Bit12 : ALIAS FOR I19[1].12;
   I19_001_Bit13 : ALIAS FOR I19[1].13;
   I19_001_Bit14 : ALIAS FOR I19[1].14;
   I19_001_Bit15 : ALIAS FOR I19[1].15;
   I1_000_Bit00 : ALIAS FOR I1[0].0;   // NIV_HOOG_VLOK1
   I1_000_Bit01 : ALIAS FOR I1[0].1;   // NIV_MID_VLOK1
   I1_000_Bit02 : ALIAS FOR I1[0].2;   // NIV_LAAG_VLOK1
   I1_000_Bit03 : ALIAS FOR I1[0].3;   // NIV_HOOG_VLOK2
   I1_000_Bit04 : ALIAS FOR I1[0].4;   // NIV_MID_VLOK2
   I1_000_Bit05 : ALIAS FOR I1[0].5;   // NIV_LAAG_VLOK2
   I1_000_Bit06 : ALIAS FOR I1[0].6;   // FC EV3
   I1_000_Bit07 : ALIAS FOR I1[0].7;   // FC EV3
   I1_000_Bit08 : ALIAS FOR I1[0].8;
   I1_000_Bit09 : ALIAS FOR I1[0].9;
   I1_000_Bit10 : ALIAS FOR I1[0].10;
   I1_000_Bit11 : ALIAS FOR I1[0].11;
   I1_000_Bit12 : ALIAS FOR I1[0].12;
   I1_000_Bit13 : ALIAS FOR I1[0].13;
   I1_000_Bit14 : ALIAS FOR I1[0].14;
   I1_000_Bit15 : ALIAS FOR I1[0].15;
   I1_001_Bit00 : ALIAS FOR I1[1].0;
   I1_001_Bit01 : ALIAS FOR I1[1].1;
   I1_001_Bit02 : ALIAS FOR I1[1].2;
   I1_001_Bit03 : ALIAS FOR I1[1].3;
   I1_001_Bit04 : ALIAS FOR I1[1].4;
   I1_001_Bit05 : ALIAS FOR I1[1].5;
   I1_001_Bit06 : ALIAS FOR I1[1].6;   // EV3 open
   I1_001_Bit07 : ALIAS FOR I1[1].7;
   I1_001_Bit15 : ALIAS FOR I1[1].15;
   I1_005_Bit0 : ALIAS FOR I1[5].0;   // Motor p 20
   I1_005_Bit1 : ALIAS FOR I1[5].1;   // Motor pd7 doseerpomp 1 floculaat
   I1_005_Bit14 : ALIAS FOR I1[5].14;
   I1_005_Bit15 : ALIAS FOR I1[5].15;
   I1_005_Bit2 : ALIAS FOR I1[5].2;   // Motor pd8 doseerpomp 2 floculaat
   I1_005_Bit3 : ALIAS FOR I1[5].3;   // Motor pomp recircuatie ingang 1 decanter
   I1_005_Bit4 : ALIAS FOR I1[5].4;   // Motor pomp pm2 recircuatie ingang 2 decanter
   I1_005_Bit5 : ALIAS FOR I1[5].5;   // Motor pomp pm3 recircuatie ingang 1 decanter
   I1_005_Bit6 : ALIAS FOR I1[5].6;   // Motor pomp pm3 recircuatie ingang 2 decanter
   I1_005_Bit7 : ALIAS FOR I1[5].7;   // res
   I1_008_Bit00 : ALIAS FOR I1[8].0;   // Noodstop gedrukt
   I1_008_Bit01 : ALIAS FOR I1[8].1;   // Hand Automaat stormbekken
   I1_008_Bit02 : ALIAS FOR I1[8].2;   // Start pomp 1 stormbekken
   I1_008_Bit03 : ALIAS FOR I1[8].3;   // Stop pomp 1 stormbekken
   I1_008_Bit04 : ALIAS FOR I1[8].4;   // Start pomp 2 stormbekken
   I1_008_Bit05 : ALIAS FOR I1[8].5;   // Stop pomp 2 stormbekken
   I1_008_Bit06 : ALIAS FOR I1[8].6;   // Start P3 stormbekken
   I1_008_Bit07 : ALIAS FOR I1[8].7;   // Stop P3 stormbekken
   I1_008_Bit08 : ALIAS FOR I1[8].8;   // Start PD1 Biocide
   I1_008_Bit09 : ALIAS FOR I1[8].9;   // Stop PD1 biocide
   I1_008_Bit10 : ALIAS FOR I1[8].10;   // start pd2 biocide
   I1_008_Bit11 : ALIAS FOR I1[8].11;   // stop pd2 biocide
   I1_008_Bit12 : ALIAS FOR I1[8].12;   // start
   I1_008_Bit13 : ALIAS FOR I1[8].13;   // stop
   I1_008_Bit14 : ALIAS FOR I1[8].14;   // freq reg biocide in bedrijf 1
   I1_008_Bit15 : ALIAS FOR I1[8].15;   // freq reg biocide in bedrijf 2
   I1_009_Bit00 : ALIAS FOR I1[9].0;   // Spanning 220 V nuts ok
   I1_009_Bit01 : ALIAS FOR I1[9].1;   // Spanning 220 v ac ok
   I1_009_Bit02 : ALIAS FOR I1[9].2;   // Spanning 24 v dc ok
   I1_009_Bit03 : ALIAS FOR I1[9].3;   // Thermische storing pomp 1
   I1_009_Bit04 : ALIAS FOR I1[9].4;   // Pomp 1 in lijn
   I1_009_Bit05 : ALIAS FOR I1[9].5;   // Pomp 1 in driehoek
   I1_009_Bit06 : ALIAS FOR I1[9].6;   // Pomp 1 in ster
   I1_009_Bit07 : ALIAS FOR I1[9].7;   // Thermische storing pomp 2
   I1_009_Bit08 : ALIAS FOR I1[9].8;   // Pomp 2 in lijn
   I1_009_Bit09 : ALIAS FOR I1[9].9;   // Pomp 2 in driehoek
   I1_009_Bit10 : ALIAS FOR I1[9].10;   // Pomp 2 in ster
   I1_009_Bit11 : ALIAS FOR I1[9].11;   // Thermische storing pomp 3
   I1_009_Bit12 : ALIAS FOR I1[9].12;   // Pomp 3 in lijn
   I1_009_Bit13 : ALIAS FOR I1[9].13;   // Pomp 3 in driehoek
   I1_009_Bit14 : ALIAS FOR I1[9].14;   // Pomp 3 in ster
   I1_009_Bit15 : ALIAS FOR I1[9].15;   // Thermische storing pomp pd1 ok
   I1_010_Bit00 : ALIAS FOR I1[10].0;   // PD1 spanning ok op regelaar
   I1_010_Bit01 : ALIAS FOR I1[10].1;   // Frequentie reg storing pd1
   I1_010_Bit02 : ALIAS FOR I1[10].2;   // Thermische storng pomp pd2 ok
   I1_010_Bit03 : ALIAS FOR I1[10].3;   // PD2 spanning ok op regelaar
   I1_010_Bit04 : ALIAS FOR I1[10].4;   // Frequentie reg storing pd2
   I1_010_Bit05 : ALIAS FOR I1[10].5;   // Vlotterschak lal stormbekken
   I1_010_Bit06 : ALIAS FOR I1[10].6;   // Storing voeding promag 33
   I1_010_Bit07 : ALIAS FOR I1[10].7;   // Inpuls promag 33 debiet
   I1_010_Bit08 : ALIAS FOR I1[10].8;   // Fout promag 33
   I1_010_Bit09 : ALIAS FOR I1[10].9;
   I1_010_Bit10 : ALIAS FOR I1[10].10;   // Noodstop relais ok stormbekken
   I1_016_Bit00 : ALIAS FOR I1[16].0;   // CL2 noodstop gedrukt
   I1_016_Bit01 : ALIAS FOR I1[16].1;   // CL2 Hamd /Autom
   I1_016_Bit02 : ALIAS FOR I1[16].2;   // CL2 start p11
   I1_016_Bit03 : ALIAS FOR I1[16].3;   // CL2 stop p11
   I1_016_Bit04 : ALIAS FOR I1[16].4;   // CL2 start p12
   I1_016_Bit05 : ALIAS FOR I1[16].5;   // CL2 stop p12
   I1_016_Bit06 : ALIAS FOR I1[16].6;   // CL2 start res.
   I1_016_Bit07 : ALIAS FOR I1[16].7;   // CL2 stop reserve
   I1_016_Bit08 : ALIAS FOR I1[16].8;   // conduc 3 kontakt 1
   I1_016_Bit09 : ALIAS FOR I1[16].9;   // conduc 3 kontakt 2
   I1_016_Bit10 : ALIAS FOR I1[16].10;   // conduc 3 alarm
   I1_016_Bit11 : ALIAS FOR I1[16].11;   // Niveau lus5 kontakt1
   I1_016_Bit12 : ALIAS FOR I1[16].12;   // Niveau lus5 kontakt2
   I1_016_Bit13 : ALIAS FOR I1[16].13;   // Niveau lus5 kontakt3
   I1_016_Bit14 : ALIAS FOR I1[16].14;   // Niveau vlotter kuip A3 lijn 3
   I1_016_Bit15 : ALIAS FOR I1[16].15;
   I1_017_Bit00 : ALIAS FOR I1[17].0;   // CL3 noodstop gedrukt
   I1_017_Bit01 : ALIAS FOR I1[17].1;   // CL3 Hamd /Autom
   I1_017_Bit02 : ALIAS FOR I1[17].2;   // CL3 start p13
   I1_017_Bit03 : ALIAS FOR I1[17].3;   // CL3 stop p13
   I1_017_Bit04 : ALIAS FOR I1[17].4;   // CL3 start p14
   I1_017_Bit05 : ALIAS FOR I1[17].5;   // CL3 stop p14
   I1_017_Bit06 : ALIAS FOR I1[17].6;   // CL3 start res.
   I1_017_Bit07 : ALIAS FOR I1[17].7;   // CL3 stop reserve
   I1_017_Bit08 : ALIAS FOR I1[17].8;   // conduc 4 kontakt 1
   I1_017_Bit09 : ALIAS FOR I1[17].9;   // conduc 4 kontakt 2
   I1_017_Bit10 : ALIAS FOR I1[17].10;   // conduc 4 alarm
   I1_017_Bit11 : ALIAS FOR I1[17].11;   // Niveau lus6 kontakt1
   I1_017_Bit12 : ALIAS FOR I1[17].12;   // Niveau lus6 kontakt2
   I1_017_Bit13 : ALIAS FOR I1[17].13;   // Niveau lus6 kontakt3
   I1_017_Bit14 : ALIAS FOR I1[17].14;   // Niveau A3 vlotter niveau
   I1_018_Bit00 : ALIAS FOR I1[18].0;   // CL4 noodstop gedrukt
   I1_018_Bit01 : ALIAS FOR I1[18].1;   // CL4 Hamd /Autom
   I1_018_Bit02 : ALIAS FOR I1[18].2;   // CL4 start p15
   I1_018_Bit03 : ALIAS FOR I1[18].3;   // CL4 stop p15
   I1_018_Bit04 : ALIAS FOR I1[18].4;   // CL4 start p16
   I1_018_Bit05 : ALIAS FOR I1[18].5;   // CL4 stop p16
   I1_018_Bit06 : ALIAS FOR I1[18].6;   // CL4 start res.
   I1_018_Bit07 : ALIAS FOR I1[18].7;   // CL4 stop reserve
   I1_018_Bit08 : ALIAS FOR I1[18].8;   // conduc 5 kontakt 1
   I1_018_Bit09 : ALIAS FOR I1[18].9;   // conduc 5 kontakt 2
   I1_018_Bit10 : ALIAS FOR I1[18].10;   // conduc 5 alarm
   I1_018_Bit11 : ALIAS FOR I1[18].11;   // Niveau lus7 kontakt1
   I1_018_Bit12 : ALIAS FOR I1[18].12;   // Niveau lus7 kontakt2
   I1_018_Bit13 : ALIAS FOR I1[18].13;   // Niveau lus7 kontakt3
   I1_018_Bit14 : ALIAS FOR I1[18].14;
   I1_018_Bit15 : ALIAS FOR I1[18].15;
   I1_019_Bit00 : ALIAS FOR I1[19].0;   // 220V ok aan lijn 123
   I2 : INT[2] := ([0] := 2#0010_0001_1111_0111, [1] := 2#0101_1101_1000_0110);
   I20 : INT[8] := ([1] := 2#0001_1001_1011_0010, [3] := 2#0011_0001_1101_1111, [5] := 2#0001_0000_1000_0010, [6] := 2#0000_1100_1100_1101, [7] := 2#0100_0000_0000_0000);
   I20_000 : ALIAS FOR I20[0];
   I20_001 : ALIAS FOR I20[1];
   I20_002 : ALIAS FOR I20[2];
   I20_003 : ALIAS FOR I20[3];
   I20_004 : ALIAS FOR I20[4];
   I20_005 : ALIAS FOR I20[5];
   I20_006 : ALIAS FOR I20[6];
   I20_007 : ALIAS FOR I20[7];
   I21 : INT[8] := ([0] := 2#0010_1001_1011_1100, [1] := 2#0001_1000_0110_0111, [2] := 2#0000_1100_1100_1110, [3] := 2#0000_1100_1100_1101, [4] := 2#0000_1100_1101_0011, [5] := 2#0000_1100_1100_1111, [6] := 2#0011_0111_1110_1001, [7] := 2#0010_1010_1101_0000);
   I21_000 : ALIAS FOR I21[0];
   I21_001 : ALIAS FOR I21[1];
   I21_002 : ALIAS FOR I21[2];
   I21_003 : ALIAS FOR I21[3];
   I21_004 : ALIAS FOR I21[4];
   I21_005 : ALIAS FOR I21[5];
   I21_006 : ALIAS FOR I21[6];
   I21_007 : ALIAS FOR I21[7];
   I22 : INT[8] := ([0] := 2#0010_0100_1001_1111, [1] := 2#0010_0000_0001_0010, [5] := 2#0001_1011_1000_0101, [7] := 2#0011_0111_1011_1101);
   I22_000 : ALIAS FOR I22[0];
   I22_001 : ALIAS FOR I22[1];
   I22_002 : ALIAS FOR I22[2];
   I22_003 : ALIAS FOR I22[3];
   I22_004 : ALIAS FOR I22[4];
   I22_005 : ALIAS FOR I22[5];
   I22_006 : ALIAS FOR I22[6];
   I22_007 : ALIAS FOR I22[7];
   I23 : INT[8] := ([0] := 2#0011_0111_0101_0110, [2] := 2#0000_1101_0010_1011, [4] := 2#0000_0100_1111_1110, [5] := 2#0011_1101_0100_0010, [6] := 2#0000_1010_1100_1011);
   I23_000 : ALIAS FOR I23[0];
   I23_001 : DINT;
   I23_002 : ALIAS FOR I23[2];
   I23_003 : ALIAS FOR I23[3];
   I23_004 : ALIAS FOR I23[4];
   I23_005 : ALIAS FOR I23[5];
   I23_006 : ALIAS FOR I23[6];
   I23_007 : DINT;
   I24 : INT[8] := ([4] := 2#0010_1100_0011_1111, [5] := 2#0010_1100_0110_0011);
   I24_000 : ALIAS FOR I24[0];
   I24_001 : ALIAS FOR I24[1];
   I24_002 : ALIAS FOR I24[2];
   I24_003 : ALIAS FOR I24[3];
   I24_004 : ALIAS FOR I24[4];
   I24_005 : ALIAS FOR I24[5];
   I24_006 : ALIAS FOR I24[6];
   I24_007 : ALIAS FOR I24[7];
   I25 : INT[8];
   I25_000 : ALIAS FOR I25[0];
   I25_001 : ALIAS FOR I25[1];
   I25_002 : ALIAS FOR I25[2];
   I25_003 : ALIAS FOR I25[3];
   I25_004 : ALIAS FOR I25[4];
   I25_005 : ALIAS FOR I25[5];
   I25_006 : ALIAS FOR I25[6];
   I25_007 : ALIAS FOR I25[7];
   I26 : INT[8] := ([0] := 2#0000_1110_1101_0010, [1] := 2#0011_1110_1001_1010, [2] := 2#0000_1100_1100_1101, [3] := 2#0011_1001_1001_0101, [4] := 2#0010_1111_1100_1001, [5] := 2#0011_0101_0100_1110, [6] := 2#0010_0101_0011_0011, [7] := 2#0001_1110_0100_1111);
   I26_000 : ALIAS FOR I26[0];
   I26_001 : ALIAS FOR I26[1];
   I26_002 : ALIAS FOR I26[2];
   I26_003 : ALIAS FOR I26[3];
   I26_004 : ALIAS FOR I26[4];
   I26_005 : ALIAS FOR I26[5];
   I26_006 : ALIAS FOR I26[6];
   I26_007 : ALIAS FOR I26[7];
   I28 : INT[8] := ([0] := 2#0010_0001_0010_0110, [1] := 2#0100_0000_0000_0000);
   I28_000 : ALIAS FOR I28[0];
   I28_001 : ALIAS FOR I28[1];
   I28_002 : ALIAS FOR I28[2];
   I28_003 : ALIAS FOR I28[3];
   I28_004 : ALIAS FOR I28[4];
   I28_005 : ALIAS FOR I28[5];
   I28_006 : ALIAS FOR I28[6];
   I28_007 : ALIAS FOR I28[7];
   I2_000_Bit00 : ALIAS FOR I2[0].0;   // Deelnoodstop cl2 lijn 1
   I2_000_Bit01 : ALIAS FOR I2[0].1;   // Deelnoodstop cl3 lijn 3
   I2_000_Bit02 : ALIAS FOR I2[0].2;   // Deelnoodstop cl4
   I2_000_Bit03 : ALIAS FOR I2[0].3;   // Deelnoodstop cl5 lijn 4
   I2_000_Bit04 : ALIAS FOR I2[0].4;   // Deelnoodstop cl6 eurowater
   I2_000_Bit05 : ALIAS FOR I2[0].5;   // Deelnoodstop cl7 IBT A
   I2_000_Bit06 : ALIAS FOR I2[0].6;   // Deelnoodstop cl7 IBT B
   I2_000_Bit07 : ALIAS FOR I2[0].7;   // Deelnoodstop cl7 IBT C
   I2_000_Bit08 : ALIAS FOR I2[0].8;   // Voeidng 220V ok
   I2_000_Bit09 : ALIAS FOR I2[0].9;   // Storing voeding lijn 1 cl 2
   I2_000_Bit10 : ALIAS FOR I2[0].10;   // Storing voeding lijn 2 cl 3
   I2_000_Bit11 : ALIAS FOR I2[0].11;   // Storing voeding lijn 3 cl 4
   I2_000_Bit12 : ALIAS FOR I2[0].12;   // Storing voeding lijn 4 cl 5
   I2_000_Bit13 : ALIAS FOR I2[0].13;   // Storing voeding lijn deel eurowater cl 6
   I2_000_Bit14 : ALIAS FOR I2[0].14;   // Storing voedingslijn IBT-A CL 7
   I2_000_Bit15 : ALIAS FOR I2[0].15;   // Storing voedingslijn IBT-B CL 8
   I2_001_Bit00 : ALIAS FOR I2[1].0;   // Storing voedingslijn IBT-C CL 9
   I2_001_Bit01 : ALIAS FOR I2[1].1;   // Voeding meting 220V ok
   I2_001_Bit02 : ALIAS FOR I2[1].2;   // Voeding DC 24 ok
   I2_001_Bit03 : ALIAS FOR I2[1].3;   // Storing voeding 24V DC algemeen
   I2_001_Bit04 : ALIAS FOR I2[1].4;   // Storing voeding 24V ingangen
   I2_001_Bit05 : ALIAS FOR I2[1].5;   // Storing 24V meting
   I2_001_Bit06 : ALIAS FOR I2[1].6;   // Voeding uitgang 24V
   I2_001_Bit07 : ALIAS FOR I2[1].7;   // Motor p11 lijn1 in dienst
   I2_001_Bit08 : ALIAS FOR I2[1].8;   // Motor p11 lijn1 thermische storing
   I2_001_Bit09 : ALIAS FOR I2[1].9;   // Motor p12 lijn1 in dienst
   I2_001_Bit10 : ALIAS FOR I2[1].10;   // Motor p12 lijn1 thermische storing
   I2_001_Bit11 : ALIAS FOR I2[1].11;   // Motor p13 lijn2 in dienst
   I2_001_Bit12 : ALIAS FOR I2[1].12;   // Motor p13 lijn2 thermische storing
   I2_001_Bit13 : ALIAS FOR I2[1].13;   // Motor p14 lijn2 in dienst
   I2_001_Bit14 : ALIAS FOR I2[1].14;   // Motor p14 lijn2 thermische storing
   I2_001_Bit15 : ALIAS FOR I2[1].15;   // Motor p15 lijn3 in dienst
   I3 : INT[2] := ([0] := 2#1000_1011_1000_0111, [1] := 2#0010_1000_1000_1000);
   I3_000_Bit00 : ALIAS FOR I3[0].0;   // Motor p15 lijn3 thermische storing
   I3_000_Bit01 : ALIAS FOR I3[0].1;   // Motor p16 lijn3 in dienst
   I3_000_Bit02 : ALIAS FOR I3[0].2;   // Motor p16 lijn3 thermische storing
   I3_000_Bit03 : ALIAS FOR I3[0].3;   // Motor p17 lijn4 in dienst
   I3_000_Bit04 : ALIAS FOR I3[0].4;   // Motor p17 lijn4 thermische storing
   I3_000_Bit05 : ALIAS FOR I3[0].5;   // Motor p18 lijn4 in dienst
   I3_000_Bit06 : ALIAS FOR I3[0].6;   // Motor p18 lijn4 thermische storing
   I3_000_Bit07 : ALIAS FOR I3[0].7;   // Motor pro 1 voedingpomp osmose 1 Thermische storing
   I3_000_Bit08 : ALIAS FOR I3[0].8;   // Motor pro 1 voedingpomp osmose 1 in lijn
   I3_000_Bit09 : ALIAS FOR I3[0].9;   // Motor pro 1 voedingpomp osmose 1 in driehoek
   I3_000_Bit10 : ALIAS FOR I3[0].10;   // Motor pro 1 voedingpomp osmose 1 in ster
   I3_000_Bit11 : ALIAS FOR I3[0].11;   // Motor pro2 voedingpomp osmose 2 Thermische storing
   I3_000_Bit12 : ALIAS FOR I3[0].12;   // Motor pro 2 voedingpomp osmose 2 in lijn
   I3_000_Bit13 : ALIAS FOR I3[0].13;   // Motor pro 2 voedingpomp osmose 2 in driehoek
   I3_000_Bit14 : ALIAS FOR I3[0].14;   // Motor pro 2 voedingpomp osmose 2 in ster
   I3_000_Bit15 : ALIAS FOR I3[0].15;   // Motor P21 Thermische storing Kuip AZ
   I3_001_Bit00 : ALIAS FOR I3[1].0;   // Motor p21 kuip az in lijn
   I3_001_Bit01 : ALIAS FOR I3[1].1;   // Motor p21 kuip az in driehoek
   I3_001_Bit02 : ALIAS FOR I3[1].2;   // Motor p21 kuip az in ster
   I3_001_Bit03 : ALIAS FOR I3[1].3;   // Thermische storing motor P22 kuip AZ
   I3_001_Bit04 : ALIAS FOR I3[1].4;   // Motor p22 kuip az in lijn
   I3_001_Bit05 : ALIAS FOR I3[1].5;   // Motor p22 kuip az in driehoek
   I3_001_Bit06 : ALIAS FOR I3[1].6;   // Motor p22 kuip az in ster
   I3_001_Bit07 : ALIAS FOR I3[1].7;   // Thermische storing motor PRO3 voedingsp. osmose 3
   I3_001_Bit08 : ALIAS FOR I3[1].8;   // Motor voedingspomp osmose 3 in lijn
   I3_001_Bit09 : ALIAS FOR I3[1].9;   // Motor voedingspomp osmose 3 in drie
   I3_001_Bit10 : ALIAS FOR I3[1].10;   // Motor voed osmose 3 ster
   I3_001_Bit11 : ALIAS FOR I3[1].11;   // Motor P21 reinigingspomp membraam
   I3_001_Bit12 : ALIAS FOR I3[1].12;   // Motor P21 reinigingspomp in dienst
   I3_001_Bit13 : ALIAS FOR I3[1].13;   // Thermische storing S2 ventilator
   I3_001_Bit14 : ALIAS FOR I3[1].14;   // Motor S2 Ventilator in diest
   I3_001_Bit15 : ALIAS FOR I3[1].15;   // Thermische storing voedingspomp fabriek 1
   I4 : INT[2] := ([0] := 2#1000_0101_0111_1000, [1] := 2#1010_1110_1011_1111);
   I4_000_Bit00 : ALIAS FOR I4[0].0;   // Motor P3 voedingspomp in lijn
   I4_000_Bit01 : ALIAS FOR I4[0].1;   // READY DRIVE P3
   I4_000_Bit02 : ALIAS FOR I4[0].2;   // defaut drive P4
   I4_000_Bit03 : ALIAS FOR I4[0].3;   // Thermische storing voedingspomp fabriek 2
   I4_000_Bit04 : ALIAS FOR I4[0].4;   // Motor p4 in lijn in
   I4_000_Bit05 : ALIAS FOR I4[0].5;   // ready drive p4
   I4_000_Bit06 : ALIAS FOR I4[0].6;   // defaut drive P4
   I4_000_Bit07 : ALIAS FOR I4[0].7;   // Motor p5 in dienst
   I4_000_Bit08 : ALIAS FOR I4[0].8;   // Thermische storing motor p 5 ok
   I4_000_Bit09 : ALIAS FOR I4[0].9;   // Motor p6 in dienst
   I4_000_Bit10 : ALIAS FOR I4[0].10;   // Thermische storing p6 ok
   I4_000_Bit11 : ALIAS FOR I4[0].11;   // pomp p23 in kelderkuip in dienst
   I4_000_Bit12 : ALIAS FOR I4[0].12;   // Thermische beveiligneing pomp p23 in kelderkuip
   I4_000_Bit13 : ALIAS FOR I4[0].13;   // Motor p24 in dienst
   I4_000_Bit14 : ALIAS FOR I4[0].14;   // Thermische beveiligneing pomp p24 in kelderkuip
   I4_000_Bit15 : ALIAS FOR I4[0].15;   // thermische storing frequentieregelaar motor p25
   I4_001_Bit00 : ALIAS FOR I4[1].0;   // spanning op freqreg motor p20
   I4_001_Bit01 : ALIAS FOR I4[1].1;   // Thermische storing freqreg p20
   I4_001_Bit02 : ALIAS FOR I4[1].2;   // Motor AG1 mixer krimp nutral in dienst
   I4_001_Bit03 : ALIAS FOR I4[1].3;   // Motor AG1 mixer vat neutral thermische st ok
   I4_001_Bit04 : ALIAS FOR I4[1].4;   // motor pd3 acide in dienst
   I4_001_Bit05 : ALIAS FOR I4[1].5;   // Motor acide thermische st ok
   I4_001_Bit06 : ALIAS FOR I4[1].6;   // motor pd4 acide in dienst
   I4_001_Bit07 : ALIAS FOR I4[1].7;   // Motor acide 4 thermische st ok
   I4_001_Bit08 : ALIAS FOR I4[1].8;   // motor pd5 soude in dienst
   I4_001_Bit09 : ALIAS FOR I4[1].9;   // Motor soude 5 thermische st ok
   I4_001_Bit10 : ALIAS FOR I4[1].10;   // motor pd6 soude in dienst
   I4_001_Bit11 : ALIAS FOR I4[1].11;   // Motor soude 6 thermische st ok
   I4_001_Bit12 : ALIAS FOR I4[1].12;   // motor ag2 mixer vat 1 voorbereiding floculaat in
   I4_001_Bit13 : ALIAS FOR I4[1].13;   // Motor ag2 mixer thermische st ok
   I4_001_Bit14 : ALIAS FOR I4[1].14;   // Motor ag3 mixer in dienst
   I4_001_Bit15 : ALIAS FOR I4[1].15;   // Motor ag3 mixer thermische st ok
   I5 : INT[2] := ([0] := 2#1111_1110_0011_1111, [1] := 2#0110_0111_0111_1111);
   I5_000_Bit00 : ALIAS FOR I5[0].0;   // thermische storing motor doseerpop1 pd7
   I5_000_Bit01 : ALIAS FOR I5[0].1;   // spanning op motor freqreg doseer floculaat
   I5_000_Bit02 : ALIAS FOR I5[0].2;   // storing freqreg doseer floculaat
   I5_000_Bit03 : ALIAS FOR I5[0].3;   // thermische storing motor freqreg doseer floculaat pd8
   I5_000_Bit04 : ALIAS FOR I5[0].4;   // spanning op motor freqreg doseer floculaat pd8
   I5_000_Bit05 : ALIAS FOR I5[0].5;   // storing freqreg doseer floculaat pd8
   I5_000_Bit06 : ALIAS FOR I5[0].6;   // pomp p19 zuiveringspomp in dienst
   I5_000_Bit07 : ALIAS FOR I5[0].7;   // thermische storing motor zuiveringspomp p19
   I5_000_Bit08 : ALIAS FOR I5[0].8;   // pomp p19b zuiveringspomp in dienst
   I5_000_Bit09 : ALIAS FOR I5[0].9;   // thermische storing motor zuiveringspomp p19b
   I5_000_Bit10 : ALIAS FOR I5[0].10;   // thermische storing motor PM1
   I5_000_Bit11 : ALIAS FOR I5[0].11;   // spanning op motor freqreg recerculatiep. dec. ingang 1
   I5_000_Bit12 : ALIAS FOR I5[0].12;   // fout freqreg recerculatiep. dec. ingang 1
   I5_000_Bit13 : ALIAS FOR I5[0].13;   // thermische storing motor recirculatiep. dec. ingang 2
   I5_000_Bit14 : ALIAS FOR I5[0].14;   // spanning freqreg. recirculatiep. dec. ingang 2
   I5_000_Bit15 : ALIAS FOR I5[0].15;   // fout freqreg recerculatiep. dec. ingang 2
   I5_001_Bit00 : ALIAS FOR I5[1].0;   // thermische storing motor evacuatiepomp dec. ingang 1
   I5_001_Bit01 : ALIAS FOR I5[1].1;   // spanning freqreg. evacuatiepomp decanter ingang 1
   I5_001_Bit02 : ALIAS FOR I5[1].2;   // fout freqreg pm3 evacuatiep. dec. ingang 1
   I5_001_Bit03 : ALIAS FOR I5[1].3;   // thermische storing motor evacuatiepomp dec. ingang 2
   I5_001_Bit04 : ALIAS FOR I5[1].4;   // spanning freqreg. evacuatiepomp decanter ingang 2
   I5_001_Bit05 : ALIAS FOR I5[1].5;   // fout freqreg pm4 evacuatiep. dec. ingang 2
   I5_001_Bit06 : ALIAS FOR I5[1].6;   // thermische storing voedingspomp 1 osmose ok
   I5_001_Bit07 : ALIAS FOR I5[1].7;   // motor pomp p7 is in dienst osmose invers
   I5_001_Bit08 : ALIAS FOR I5[1].8;   // thermische storing voedingspomp 2 osmose ok
   I5_001_Bit09 : ALIAS FOR I5[1].9;   // motor pomp p8 is in dienst osmose invers
   I5_001_Bit10 : ALIAS FOR I5[1].10;   // thermische storing voedingspomp 3 osmose ok
   I5_001_Bit11 : ALIAS FOR I5[1].11;   // motor pomp p9 is in dienst osmose invers
   I5_001_Bit12 : ALIAS FOR I5[1].12;   // EV6_OPEN
   I5_001_Bit13 : ALIAS FOR I5[1].13;   // EV6_TOE
   I5_001_Bit14 : ALIAS FOR I5[1].14;   // EV7_TOE
   I5_001_Bit15 : ALIAS FOR I5[1].15;   // EV7_OPEN
   I6 : INT[2] := ([0] := 2#1001_1100_0001_0000, [1] := 2#0010_0011_0110_0000);
   I6_000_Bit00 : ALIAS FOR I6[0].0;   // totaal debiet tfb1
   I6_000_Bit01 : ALIAS FOR I6[0].1;   // totaal debiet stfa 2
   I6_000_Bit02 : ALIAS FOR I6[0].2;   // totaal 3 debiet stfa 3
   I6_000_Bit03 : ALIAS FOR I6[0].3;   // TH pmp PUT 2
   I6_000_Bit04 : ALIAS FOR I6[0].4;   // TH PMP PUT over
   I6_000_Bit05 : ALIAS FOR I6[0].5;   // th PMP PUT 1
   I6_000_Bit06 : ALIAS FOR I6[0].6;   // non existant th pmp 1 vijver
   I6_000_Bit07 : ALIAS FOR I6[0].7;   // pulsteller debiet ontijzer 2
   I6_000_Bit08 : ALIAS FOR I6[0].8;   // hardheidsmeting kontakt 1
   I6_000_Bit09 : ALIAS FOR I6[0].9;   // hardheidsmeting kontakt 2
   I6_000_Bit10 : ALIAS FOR I6[0].10;   // pressostaat osmose1
   I6_000_Bit11 : ALIAS FOR I6[0].11;   // pressostaat osmose2
   I6_000_Bit12 : ALIAS FOR I6[0].12;   // pressostaat osmose3
   I6_000_Bit13 : ALIAS FOR I6[0].13;   // ES_EV2_IS_TOE
   I6_000_Bit14 : ALIAS FOR I6[0].14;   // ES_EV2_IS_OPEN
   I6_000_Bit15 : ALIAS FOR I6[0].15;   // Lus 1 niveau reservoir kontakt 3
   I6_001_Bit00 : ALIAS FOR I6[1].0;   // hoog alarm ketel pretraitec water
   I6_001_Bit01 : ALIAS FOR I6[1].1;   // Lus 1 niveau ketel hoog
   I6_001_Bit02 : ALIAS FOR I6[1].2;   // laag alarm pretraitec water
   I6_001_Bit03 : ALIAS FOR I6[1].3;   // zeer laag alarm pretraitec water
   I6_001_Bit04 : ALIAS FOR I6[1].4;   // niveau silo disolvent
   I6_001_Bit05 : ALIAS FOR I6[1].5;   // debietsmeting q2 pulsen
   I6_001_Bit06 : ALIAS FOR I6[1].6;   // debietsmeting q2 fout 1
   I6_001_Bit07 : ALIAS FOR I6[1].7;   // pulse debietmeter zandfilter osmose
   I6_001_Bit08 : ALIAS FOR I6[1].8;   // debietsmeting q3 pulsen
   I6_001_Bit09 : ALIAS FOR I6[1].9;   // debietsmeting q3 fout 1
   I6_001_Bit10 : ALIAS FOR I6[1].10;   // debietsmeting q3 fout 2
   I6_001_Bit11 : ALIAS FOR I6[1].11;   // Ph meting vervuild water kontakt 1
   I6_001_Bit12 : ALIAS FOR I6[1].12;   // Ph meting vervuild water fout
   I6_001_Bit13 : ALIAS FOR I6[1].13;   // ph1.2. vervuild water kontakt 1
   I6_001_Bit14 : ALIAS FOR I6[1].14;   // ph 1.2 meting puls
   I6_001_Bit15 : ALIAS FOR I6[1].15;   // meting recup water kontakt 1
   I7 : INT[2] := ([0] := 2#1100_0000_0111_1110, [1] := 2#0000_0011_1001_1111);
   I7_000_Bit00 : ALIAS FOR I7[0].0;   // ph meting fout gerecycleerd water
   I7_000_Bit01 : ALIAS FOR I7[0].1;   // lus2 niveau kontakt 1
   I7_000_Bit02 : ALIAS FOR I7[0].2;   // lus2 niveau kontakt 2
   I7_000_Bit03 : ALIAS FOR I7[0].3;   // lus2 niveau kontakt 3
   I7_000_Bit04 : ALIAS FOR I7[0].4;   // lus3 niveau kontakt 1
   I7_000_Bit05 : ALIAS FOR I7[0].5;   // lus3 niveau kontakt 2
   I7_000_Bit06 : ALIAS FOR I7[0].6;   // lus3 niveau kontakt 3
   I7_000_Bit07 : ALIAS FOR I7[0].7;   // hoog alarm ketel tampon
   I7_000_Bit08 : ALIAS FOR I7[0].8;   // midden alarm ketel tampon
   I7_000_Bit09 : ALIAS FOR I7[0].9;   // laag alarm ketel tampon
   I7_000_Bit10 : ALIAS FOR I7[0].10;   // zeer hoog alarm ketel clarifee
   I7_000_Bit11 : ALIAS FOR I7[0].11;   // hoog zeer hoog alarm ketel clarifee
   I7_000_Bit12 : ALIAS FOR I7[0].12;   // laag alarm ketel clarifee
   I7_000_Bit13 : ALIAS FOR I7[0].13;   // zeer laag alarm ketel clarifee
   I7_000_Bit14 : ALIAS FOR I7[0].14;   // lus 4 niveau ketel clarifiee kontakt 1
   I7_000_Bit15 : ALIAS FOR I7[0].15;   // lus 4 niveau ketel clarifiee kontakt 2
   I7_001_Bit00 : ALIAS FOR I7[1].0;   // lus 4 niveau ketel clarifiee kontakt 3
   I7_001_Bit01 : ALIAS FOR I7[1].1;   // Conductiviteit 1 kontakt 1
   I7_001_Bit02 : ALIAS FOR I7[1].2;   // Conductiviteit 1 kontakt 2
   I7_001_Bit03 : ALIAS FOR I7[1].3;   // Conductiviteit 1 alarm 3
   I7_001_Bit04 : ALIAS FOR I7[1].4;   // Conductiviteit 2 kontakt 1
   I7_001_Bit05 : ALIAS FOR I7[1].5;   // Conductiviteit 2 kontakt 2
   I7_001_Bit06 : ALIAS FOR I7[1].6;   // Conductiviteit 2 kontakt alarm
   I7_001_Bit07 : ALIAS FOR I7[1].7;   // q4 inpulsen osmose globaal
   I7_001_Bit08 : ALIAS FOR I7[1].8;   // q4 debietsmeting osmose 1 fout
   I7_001_Bit09 : ALIAS FOR I7[1].9;   // q4 debietsmeting osmose 1 fout 2
   I7_001_Bit10 : ALIAS FOR I7[1].10;   // conductiviteit kontakt 1
   I7_001_Bit11 : ALIAS FOR I7[1].11;   // Lus 8 niveau kontakt 2
   I7_001_Bit12 : ALIAS FOR I7[1].12;   // Lus 8 niveau kontakt 3
   I7_001_Bit13 : ALIAS FOR I7[1].13;   // lus 8 niveau kontakt 1
   I7_001_Bit14 : ALIAS FOR I7[1].14;   // lus 8 niveau kontakt 2
   I7_001_Bit15 : ALIAS FOR I7[1].15;   // lus 8 niveau kontakt 3
   I8 : INT[2] := ([0] := 2#0000_0000_0000_0110, [1] := 2#1010_1010_0000_0000);
   I8_000_Bit00 : ALIAS FOR I8[0].0;   // niveau kuip az hoog alarm
   I8_000_Bit01 : ALIAS FOR I8[0].1;   // niveau kuip az midden
   I8_000_Bit02 : ALIAS FOR I8[0].2;   // niveau kuip az laag niv
   I8_000_Bit03 : ALIAS FOR I8[0].3;   // niveau kuip az zeer laag niv alarm
   I8_000_Bit04 : ALIAS FOR I8[0].4;   // niveau kuip 20m hoog alarm
   I8_000_Bit05 : ALIAS FOR I8[0].5;   // niveau midden kuip 20m
   I8_000_Bit06 : ALIAS FOR I8[0].6;   // niveau kuip 20m laag niv
   I8_000_Bit07 : ALIAS FOR I8[0].7;   // niveau laag alarm curve a2
   I8_000_Bit08 : ALIAS FOR I8[0].8;   // laag niveau kuip 1 voorb. polyelectrolute
   I8_000_Bit09 : ALIAS FOR I8[0].9;   // midden niveau kuip 1 voorb. polyelectrolute
   I8_000_Bit10 : ALIAS FOR I8[0].10;   // hoog niveau kuip 1 voorb. polyelectrolute
   I8_000_Bit11 : ALIAS FOR I8[0].11;   // hoog niveau kuip 2 voorb. polyelectrolute
   I8_000_Bit12 : ALIAS FOR I8[0].12;   // midden niveau kuip 2 voorb. polyelectrolute
   I8_000_Bit13 : ALIAS FOR I8[0].13;   // hoog niveau pekel
   I8_000_Bit14 : ALIAS FOR I8[0].14;
   I8_000_Bit15 : ALIAS FOR I8[0].15;
   I8_001_Bit00 : ALIAS FOR I8[1].0;   // cl5 noodstop gedrukt
   I8_001_Bit01 : ALIAS FOR I8[1].1;   // hand automaat cl5
   I8_001_Bit02 : ALIAS FOR I8[1].2;   // drukknop start cl5 p17
   I8_001_Bit03 : ALIAS FOR I8[1].3;   // drukknop stop cl5 p17
   I8_001_Bit04 : ALIAS FOR I8[1].4;   // drukknop start cl5 p18
   I8_001_Bit05 : ALIAS FOR I8[1].5;   // drukknop stop cl5 p18
   I8_001_Bit06 : ALIAS FOR I8[1].6;   // drukknop start cl5 res
   I8_001_Bit07 : ALIAS FOR I8[1].7;   // drukknop stop cl5 res
   I8_001_Bit08 : ALIAS FOR I8[1].8;   // cl6 noodstop gedrukt
   I8_001_Bit09 : ALIAS FOR I8[1].9;   // Schakelaar hand autom cl6
   I8_001_Bit10 : ALIAS FOR I8[1].10;   // drukknop start cl6 pro1
   I8_001_Bit11 : ALIAS FOR I8[1].11;   // drukknop stop cl6 pro1
   I8_001_Bit12 : ALIAS FOR I8[1].12;   // drukknop start cl6 pro2
   I8_001_Bit13 : ALIAS FOR I8[1].13;   // drukknop stop cl6 pro2
   I8_001_Bit14 : ALIAS FOR I8[1].14;   // drukknop start cl6 p21
   I8_001_Bit15 : ALIAS FOR I8[1].15;   // drukknop stop cl6 p21
   I9 : INT[2] := ([0] := 2#1010_1010_1010_1010, [1] := 2#1010_1010_1010_1010);
   I9_000_Bit00 : ALIAS FOR I9[0].0;   // Drukknop start CL6 P22
   I9_000_Bit01 : ALIAS FOR I9[0].1;   // Drukknop stop CL6 P22
   I9_000_Bit02 : ALIAS FOR I9[0].2;   // Drukknop start CL6 PRO3
   I9_000_Bit03 : ALIAS FOR I9[0].3;   // Drukknop stop CL6 PRO3
   I9_000_Bit04 : ALIAS FOR I9[0].4;   // Drukknop start CL6 P21
   I9_000_Bit05 : ALIAS FOR I9[0].5;   // Drukknop stop CL6 P21
   I9_000_Bit06 : ALIAS FOR I9[0].6;   // Drukknop start CL6 S1
   I9_000_Bit07 : ALIAS FOR I9[0].7;   // Drukknop stop CL6 S1
   I9_000_Bit08 : ALIAS FOR I9[0].8;   // Noodstop CL7 gedrukt
   I9_000_Bit09 : ALIAS FOR I9[0].9;   // Hand_Auto CL7
   I9_000_Bit10 : ALIAS FOR I9[0].10;   // Drukknop start CL7 P3
   I9_000_Bit11 : ALIAS FOR I9[0].11;   // Drukknop stop CL7 P3
   I9_000_Bit12 : ALIAS FOR I9[0].12;   // Drukknop start CL7 P4
   I9_000_Bit13 : ALIAS FOR I9[0].13;   // Drukknop stop CL7 P4
   I9_000_Bit14 : ALIAS FOR I9[0].14;   // Drukknop start CL7 P5
   I9_000_Bit15 : ALIAS FOR I9[0].15;   // Drukknop stop CL7 P5
   I9_001_Bit00 : ALIAS FOR I9[1].0;   // Drukknop start CL7 P6
   I9_001_Bit01 : ALIAS FOR I9[1].1;   // Drukknop stop CL7 P6
   I9_001_Bit02 : ALIAS FOR I9[1].2;   // Drukknop start CL7 P23
   I9_001_Bit03 : ALIAS FOR I9[1].3;   // Drukknop stop CL7 P23
   I9_001_Bit04 : ALIAS FOR I9[1].4;   // Drukknop start CL7 P24
   I9_001_Bit05 : ALIAS FOR I9[1].5;   // Drukknop stop CL7 P24
   I9_001_Bit06 : ALIAS FOR I9[1].6;   // Drukknop start CL7 AG1
   I9_001_Bit07 : ALIAS FOR I9[1].7;   // Drukknop stop CL7 AG1
   I9_001_Bit08 : ALIAS FOR I9[1].8;   // Drukknop start CL7 AG2
   I9_001_Bit09 : ALIAS FOR I9[1].9;   // Drukknop stop CL7 AG2
   I9_001_Bit10 : ALIAS FOR I9[1].10;   // Drukknop start CL7 AG3
   I9_001_Bit11 : ALIAS FOR I9[1].11;   // Drukknop stop CL7 AG3
   I9_001_Bit12 : ALIAS FOR I9[1].12;   // Drukknop start CL7 A
   I9_001_Bit13 : ALIAS FOR I9[1].13;   // Drukknop stop CL7 pd7
   I9_001_Bit14 : ALIAS FOR I9[1].14;   // drukknop start cl7 pd8
   I9_001_Bit15 : ALIAS FOR I9[1].15;   // drukknop stop cl7 pd8
   ibt_level_soude_plein : BOOL := 1;
   ibtlancy1 : DINT := 48;
   inb : DINT := -1481572010;
   INT_COND_KOEL : integrat := (rate := 500, oai := 3802, AI := 3784);
   int_flw_put3 : integrat := (rate := 15, oai := -30, AI := -30);
   INT_LVL_KOEL : integrat := (rate := 200, oai := 857, AI := 858);
   KRK_K1 : REAL := 215.36966;
   KRK_K2 : DINT := 296;
   L1_stat : DINT[20] := ([1] := -32752, [3] := 336, [5] := 509, [6] := -32474, [9] := 1, [13] := 16, [19] := 190);
        [13].4   // fc vanne nitrique fermée
        [13].2   // fc vanne nitrique ouverte
        [13].3   // L1 ok pour fill up
        [13].1   // Bp arret de superv
        [13].0   // Bp demande Nitrique
        [3].0   // DE PLC L1demande acide
        [3].2   // de plc ligne 1fc vanne acideano ouv
        [3].4   // de plc ligne 1fc vanne acideano ferme
        [3].5   // de plc ligne 1fc vanne acideneut ouv
        [3].6   // de plc ligne 1fc vanne acideneut ferme
        [3].7   // de plc ligne 1fc vanne acidecolo ouv
        [3].8   // de plc ligne 1fc vanne acidecolo fermé
        [13].5   // lvl neutral trop haut
        [0].0   // jbk
        [4].0   // nvk
        [5].0   // fchgjhgk
        [0]   // quantité soude demandee
        [1].0   // vers plc stock demande de soude L2
        [1].1   // vers plc stock demande d'arret apport soude
        [1].2   // vers plc stock fc vanne apport soude décapage open
        [1].3   // vers plc stock apport soude finit
        [1].4   // vers plc stock fc vanne apport soudefermee
        [1].15   // T°COLMATAGE <95°
        [2]   // quantité acide demandee
        [2].0   // ghvjh
        [2].1   // vers plc stock demande d'arret apport acide
        [2].2   // vers plc stock fc vanne apport acide open
        [2].3   // vers plc stock apport acide finit
        [2].4   // vers plc stock fc vanne apport acid fermee
        [2].5   // fc vanne apport acide neutral open
        [2].6   // fc vanne apport acide neutral close
   L2_L3_OK : BOOL := 1;
   L2_L3_ppas : DINT := 5;
   L2_STAT : DINT[20] := ([1] := 4112, [2] := 80, [5] := 346, [6] := 1062, [8] := 4, [9] := -12, [11] := 10, [12] := 500, [13] := 16);
        [13].2   // fc vanne nitrique ouverte
        [13].4   // fc vanne nitrique fermee
        [13].5   // lvl Neutral trop haut
        [1].12   // de line 2line 2 run
   l2va2 : BOOL := 1;
   l2va3 : BOOL;
   L3_STAT : DINT[20] := ([0] := 100, [1] := 32784, [2] := 80, [5] := 484, [6] := 430, [8] := 4, [9] := -1, [11] := 10, [13] := 4);
        [13].4   // fc vanne nitrique fermée
        [13].2   // fc vanne nitrique ouverte
        [13].0   // Bp demande Nitrique
        [13].1   // Bp arret de superv
        [13].3   // L3 ok pour fill up
        [13].5   // lvl neutral trop haut
        [0]   // quantité soude demandee
        [1].0   // vers plc stock demande de soude L3
        [1].1   // vers plc stock demande d'arret apport soude
        [1].2   // vers plc stock fc vanne apport soude décapage open
        [1].3   // vers plc stock apport soude finit
        [1].4   // vers plc stock fc vanne apport soudefermee
        [1].15   // T°COLMATAGE <95°
        [2]   // quantité acide demandee
        [2].0   // vers plc stock demande de acide
        [2].1   // vers plc stock demande d'arret apport acide
        [2].2   // vers plc stock fc vanne apport acide open
        [2].3   // vers plc stock apport acide finit
        [2].4   // vers plc stock fc vanne apport acid fermee
        [2].5   // fc vanne apport acide neutral open
        [2].6   // fc vanne apport acide neutral close
        [3].0   // DEMANDE ACIDE
        [3].1   // DEMENDE ARRET ACIDE
   l3va1 : BOOL;
   l3va2 : BOOL := 1;
   l3va3 : BOOL;
   l3va4 : BOOL;
   L4_R2_3_O : BOOL;
   lancyibt1 : DINT;
   lancystock1 : DINT;
   lancystock2 : DINT := 16;
   lastmonth_h2so4_L1 : DINT := 6975;
   lastmonth_h2so4_L2 : DINT := 4941;
   lastmonth_h2so4_L3 : DINT := 10574;
   lastmonth_h2so4_L4 : DINT;
   lastmonth_h2so4_stat : REAL;
   lastmonth_naoh_L1 : DINT := 5959;
   lastmonth_naoh_L2 : DINT := 2942;
   lastmonth_naoh_L3 : DINT := 2805;
   lastmonth_naoh_L4 : DINT;
   lastmonth_naoh_stat : DINT := 2158;
   lastmonth_put1 : DINT := 62668;
   lastmonth_put2 : DINT := 171882;
   lastmonth_totosmose : DINT := 305607;
   lastmonth_totq1 : DINT := 778057;
   lastmonth_totq2 : DINT := 808852;
   lastmonth_totq3 : DINT := 603673;
   LDN_L1 : DINT := 333;
   LDN_L2 : REAL := 165.10109;
   LDN_L3 : REAL := 241.76395;
   LVL_AZ : REAL := 78.85;
   LVL_LUS2_ACIDE : REAL := 838.5595;
   LVL_LUS3_NAOH : REAL := 830.7774;
   LVL_NITRIC : REAL := 1327.5349;
   LVL_PRETRAITEMENT : REAL := 84.11536;
   LVL_PUISARD_IBT : DINT := 252;
   LVL_PUISARD_L4 : REAL := -25.001907;
   LVL_ZOUT : REAL := -25.001907;
   mem1 : REAL := 0.34375;
   mem3 : REAL := 0.640625;
   mem_vent_yesterdsay : REAL := 5745236.0;
   mem_water_flow_to_l1 : REAL := 139763.62;
   mem_water_flow_to_l2 : REAL := 90148.086;
   mem_water_flow_to_l3 : DINT := 35;
   mem_water_flow_to_l31 : REAL := 205436.05;
   memjour : DINT := 20;
   memo_flow_l1 : REAL := 129612.945;
   memo_flow_l2 : REAL := 84089.73;
   memo_flow_l3 : REAL := 192451.31;
   memventyesterdsay : EIGHT_POS_MODE_SELECTOR;
   MinorFaultBits : DINT;   // MinorFaultBits
   MSG_R_L2 : MESSAGE;
        MessageParameters(ServiceCode := 16#0fa2, LocalElement := N[105], ...)
   MSG_R_L3 : MESSAGE;
        MessageParameters(ServiceCode := 16#0fa2, LocalElement := N[145], ...)
   MSG_R_L4 : MESSAGE;
        MessageParameters(ServiceCode := 16#0f68, LocalElement := N[185], ...)
   MSG_R_Lancy2 : MESSAGE;
        MessageParameters(ServiceCode := 16#0fa2, LocalElement := N[225], ...)
   msg_W_L2 : MESSAGE;
        MessageParameters(ServiceCode := 16#0faa, LocalElement := N[125], ...)
   msg_W_L3 : MESSAGE;
        MessageParameters(ServiceCode := 16#0faa, LocalElement := N[165], ...)
   MSG_W_L4 : MESSAGE;
        MessageParameters(ServiceCode := 16#0f67, LocalElement := N[205], ...)
   msg_W_lancy : MESSAGE;
        MessageParameters(ServiceCode := 16#0faa, LocalElement := N7[20], ...)
   msg_W_lancy2 : MESSAGE;
        MessageParameters(ServiceCode := 16#0faa, LocalElement := N[20], ...)
   msg_W_lancy3 : MESSAGE;
        MessageParameters(ServiceCode := 16#0faa, LocalElement := N[245], ...)
   MW : BOOL := 1;
   MW1 : BOOL;
   mw2 : BOOL;
   mwcsth : DINT := 492;
   mwcsthh : DINT := 512;
   mwcstl : DINT := 485;
   mwcstll : DINT := 482;
   N : INT[255] := ([1] := -3486, [3] := 2, [10] := 61, [20] := 26, [21] := 8, [22] := 3, [40] := 10, [42] := -4, [43] := -1, [66] := 225, [69] := 5, [72] := 84, [73] := 84, [86] := 416, [87] := -30336, [108] := 82, [126] := 288, [128] := 150, [131] := 16, [133] := 336, [172] := 3488, [174] := -30336, [186] := 16, [188] := 16, [208] := 1000, [209] := 1, [226] := 16, [227] := 14, [228] := -75, [245] := 88, [252] := 3488, [254] := -30336);
        [2]   // flow acide
        [10].0   // stock acide pas haut
        [10].1   // stock acide pas bas
        [10].2   // stock mazout pashaut
        [10].3   // stock mazout pas bas
        [10].4   // stock soude L1 pashaut
        [10].5   // stock soude L1 pasbas
        [10].7   // stock soude L2 pasbas
        [10].8   // stock soude L3 pashaut
        [10].9   // stock soude L3 pasbas
        [10].10   // PVvanne soude L1fermée
        [10].13   // de PVchargement en cours
        [10].14   // DE PVBP EV SOUDE L1
        [11].0   // DE PVBP EV SOUDE L3
        [11].1   // vers PVfuite stock acide
        [11].2   // vers PVfuite stock mazout
        [11].3   // fuite soude
        [15]   // T° ambiantecabine RED L1
        [16]   // conductivité en µS
        [17]   // niveau eautour refroidissement
        [18]   // total eau tour L1 2
        [20].0   // NAOHL1 VA4FC O
        [20].1   // NAOHL1 VA4FC F
        [20].2   // NAOHL2 VA4FC O
        [20].3   // NAOHL2 VA4FC F
        [30]   // MESSAGE TO LANCY
        [46].2   // DE PLC 1VANNE SOUDEL1 OUVERTE
        [50]   // communication avecplc L1 read
        [65]   // quantité soudedemandée L1
        [66].0   // DE PLC L1demande soudeL1
        [66].1   // DE PLC L1demandearret soude L1
        [66].2   // de plc ligne 1fc vanne soudeouverte
        [66].3   // de plc ligne 1apport soudefinit
        [66].4   // de plc ligne 1fc vanne soudefermée
        [66].15   // de line 1line 1 run
        [67]   // quantité acidedemandée L1
        [67].0   // DE LANCY OPEN L1VA4
        [67].1   // DE LANCY OPEN L2VA4
        [68].1   // DE PLC L1demandearret acide L1
        [68].2   // de plc ligne 1fc vanne acideano ouv
        [68].3   // de plc ligne 1apport acidefinit
        [68].4   // de plc ligne 1fc vanne acideano ferme
        [68].5   // de plc ligne 1fc vanne acideneut ouv
        [70]   // communication avecplc L1 write
        [71]   // N:71
        [85]   // quantité souderestante L1
        [86].0   // vers plc l1 fuiteacide
        [86].1   // vers plc l1fuite soude
        [86].2   // vers plc L1fuite mazout
        [86].3   // vers plc L1ouvrir vannesoude
        [86].4   // vers plc L1apport soudefinit L1
        [86].5   // vers plc L1apport soudeoccupé
        [86].6   // vers plc L1apport soudeL1 accordé
        [86].7   // VERS PLC L1SOUDE VERS L1
        [86].8   // VERS PLC L1SOUDE VERS L2
        [86].9   // VERS PLC L1SOUDE VERS L3
        [86].10   // VERS PLC L1SOUDE VERS L4
        [86].11   // VERS PLC L1SOUDE VERS STAT
        [86].12   // DEFAULT FLOW TO L1VERS SLC
        [87]   // vers plc L1
        [87].3   // vers plc L1ouvrir vanneacide
        [87].4   // vers plc L1apport acidefinit L1
        [87].5   // vers plc L1apport acideoccupé
        [87].6   // vers plc L1apport acideaccordé
        [87].7   // VERS PLC L1acide VERS ano L1
        [87].8   // VERS PLC L1acideVERS L2
        [87].9   // VERS PLC L1acide VERS L3
        [87].10   // VERS PLC L1acide VERS L4
        [87].11   // VERS PLC L1acide VERS neutralL1
        [87].12   // VERS PLC L1 acideneutralL2
        [87].13   // VERS PLC L1acide neutralL3
        [87].14   // VERS PLC L1 acide VEL4
        [88]   // quantité aciderestante L1
        [90]   // communication avecplc L2 read
        [97]   // ?
        [98]   // ?
        [105]   // quantité soudedemandée L2
        [106].0   // DE PLC L2demande soudeL2
        [106].1   // DE PLC L2demandearret soude
        [106].2   // de plc ligne 2fc vanne soudeouverte
        [106].4   // de plc ligne 2fc vanne soudefermée
        [106].15   // de line 2line 2 run
        [107]   // quantité acidedemandée L2
        [108].0   // DE PLC L2demande acide
        [108].1   // DE PLC L2demandearret acide L2
        [108].2   // de plc ligne 2fc vanne acideouverte
        [108].4   // de plc ligne 2fc vanne acidefermée
        [108].5   // de plc ligne 2fc vanne acideneutral ouv
        [108].6   // de plc ligne 2fc vanne acideneutral ferm
        [110]   // communication avecplc L2 write
        [111]   // HULPWOORD_N1
        [112]   // HULPWOORD_N2
        [113]   // HULPWOORD_N3
        [114]   // HULPWOORD_N4
        [115]   // HULPWOORD_N5
        [125]   // quantité souderestante L2
        [126].3   // vers plc L2ouvrir vannesoude
        [126].4   // vers plc L2apport soudefinit L2
        [126].5   // vers plc L2apport soudeoccupé
        [126].6   // vers plc L2apport soudeL2 accordé
        [126].7   // VERS PLC L2SOUDE VERS L1
        [126].8   // VERS PLC L2SOUDE VERS L2
        [126].9   // VERS PLC L2SOUDE VERS L3
        [126].10   // VERS PLC L2SOUDE VERS L4
        [126].11   // VERS PLC L2SOUDE VERS STAT
        [126].12   // DEFAULT FLOW TO L2VERS SLC
        [127].3   // vers plc L2ouvrir vanneacide
        [127].4   // vers plc L2apport acidefinit L2
        [127].5   // vers plc L2apport acideoccupé
        [127].6   // vers plc L2apport acideaccordé
        [127].7   // VERS PLC L2acide VERS ano L1
        [127].8   // VERS PLC L2acide VERS L2
        [127].9   // VERS PLC L2acide VERS L3
        [127].10   // VERS PLC L2acide VERS L4
        [127].11   // VERS PLC L2acide VERS neutralL1
        [127].12   // VERS PLC L2 acideneutralL2
        [127].13   // VERS PLC L2 acideneutralL3
        [127].14   // VERS PLC L2 acide VEL4
        [128]   // quantite acidepassé l2
        [130]   // communication L3read
        [139]   // MEMODEFAUT DEGRAISSAGE
        [145]   // quantité soudedemandéel3
        [146].0   // DE PLC L3demande soudeL3
        [146].1   // DE PLC L3demandearret soude L3
        [146].2   // de plc ligne 3fc vanne soudeouverte
        [146].4   // de plc ligne 3fc vanne soudefermée
        [146].15   // ligne 3 runcolmatage
        [147]   // quantité acidedemandée l3
        [148].0   // DE PLC L3demande acide L3
        [148].1   // DE PLC L3demandearret acide L3
        [148].2   // de plc ligne 3fc vanneacide ouverte
        [148].4   // de plc ligne 3fc vanne acidefermée
        [148].5   // de plc ligne 3fc vanneacide neutral ouv
        [148].6   // de plc ligne 3fc vanneacide neutral ferm
        [150]   // communication L3write
        [165]   // quantité souderestante L3
        [166].3   // vers plc L3ouvrir vannesoude
        [166].4   // vers plc L3apport soudeL3 finit
        [166].5   // vers plc L3apport soudeoccupé
        [166].6   // vers plc L3apport soudeL3 accordé
        [166].7   // VERS PLC L3SOUDE VERS L1
        [166].8   // VERS PLC L3SOUDE VERS L2
        [166].9   // VERS PLC L3SOUDE VERS L3
        [166].10   // VERS PLC L3SOUDE VERS L4
        [166].11   // VERS PLC L3SOUDE VERS STAT
        [166].12   // DEFAULT FLOW TO L3VERS SLC
        [167].3   // vers plc L3ouvrir vanneacide
        [167].4   // vers plc L3apport acidefinit L3
        [167].5   // apport acide occupé
        [167].6   // apport acide accordé
        [167].7   // VERS PLC L3acide VERS ano L1
        [167].8   // VERS PLC L3acide VERS L2
        [167].9   // VERS PLC L3acide VERS L3
        [167].10   // VERS PLC L4acide VERS L4
        [167].11   // VERS PLC L3acide VERS neutralL1
        [167].12   // VERS PLC L3 acideneutralL2
        [167].13   // VERS PLC L3acideneutral L3
        [167].14   // VERS PLC L3 acide VEL4
        [168]   // quantite acidepassé l3
        [170]   // communicationL4
        [185]   // quantité soudedemandéel4
        [186].0   // DE PLC L4demande soudeL4
        [186].1   // DE PLC L4demandearret soude l4
        [186].2   // de plc ligne 4fc vanne soudeouverte
        [186].4   // de plc ligne 4fc vanne soudefermée
        [187]   // quantité acidedemandée L4
        [188].0   // DE PLC L4demande acide
        [188].1   // DE PLC L4demandearret acide L4
        [188].2   // de plc ligne 4fc vanne acideouverte
        [188].4   // de plc ligne 3fc vanne acidefermée
        [188].5   // de plc ligne 4fc vanne acideneutral ouv
        [188].6   // de plc ligne 4fc vanne acideneutral ferme
        [190]   // communicationL4
        [191]   // defaut niv 2
        [197]   // NOMBRE DEFAUT EXISTANT ACQUITE
        [198]   // NOMBRE NOUVEAU DEFAUT
        [199].0   // arret entretien
        [199].1   // acquit defaut
        [199].5   // new defaut
        [199].6   // ancien defaut present
        [200].0   // PMP ETANG EN DEF
        [200].1   // no flow pumping from etang
        [200].2   // FLOW TOO LOW Q1
        [200].3   // LEVEL PRETREATED TOO HIGH
        [200].4   // LEVEL LOW PRETREATED WATER WARNING
        [200].5   // LEVEL LOW PRETREATED WATER
        [200].6   // ANORMAL EMPTYING PRETREATED WATER TANK
        [200].7   // 2 pump pretreated tank out of order P3&P4
        [200].8   // no flow pumping from PRETREATED WATER TANK
        [200].9   // FLOW TOO LOW Q2
        [200].11   // recup water tank L1 too high
        [200].12   // PMP RECUP L1 OUT OF ORDER
        [200].13   // recup water tank L2 too high
        [200].14   // PMP RECUP L2 OUT OF ORDER
        [200].15   // recup water tank L3 too high
        [201].0   // PMP RECUP L3 OUT OF ORDER
        [201].1   // recup water tank L4 too high
        [201].2   // PMP RECUP L4 OUT OF ORDER
        [201].3   // LEVEL NAOH TOO HIGH
        [201].4   // ANORMAL LEVEL DECREASE naoh TANK
        [201].5   // LACK DETECTIE NAOH
        [201].6   // LEVEL H2SO4 TOO HIGH
        [201].7   // ANORMAL LEVEL DECREASE H2SO4 TANK
        [201].8   // LACK DETECTIE H2SO4
        [201].9   // defaut niveau vijver trop bas
        [201].10   // defaut niveau puisard ligne 4
        [201].11   // defaut vanne position eau ville
        [205]   // quantité souderestante L4
        [206].3   // vers plc L4ouvrir vannesoude
        [206].4   // vers plc L4apport soudeL4 finit
        [206].5   // vers plc L4apport soudeoccupé
        [206].6   // vers plc L4apport soudeL4 accordé
        [206].7   // VERS PLC L4SOUDE VERS L1
        [206].8   // VERS PLC L4SOUDE VERS L2
        [206].9   // VERS PLC L4SOUDE VERS L3
        [206].10   // VERS PLC L4SOUDE VERS L4
        [206].11   // VERS PLC L4SOUDE VERS STAT
        [207].3   // vers plc L4ouvrir vanneacide
        [207].4   // vers plc L4apport acidefinit L4
        [207].5   // vers plc L4apport acideoccupé
        [207].6   // vers plc L4apport acideaccordé
        [207].7   // VERS PLC L4acide VERS ano L1
        [207].8   // VERS PLC L4acide VERS L2
        [207].9   // VERS PLC L4acide VERS L3
        [207].10   // VERS PLC L4acide VERS L4
        [207].11   // VERS PLC L4acide VERS neutralL1
        [207].12   // VERS PLC L4 acideneutralL2
        [207].13   // VERS PLC L4acide neutralL3
        [207].14   // VERS PLC L4 acide VEL4
        [208]   // quantite acidepassé l4
        [210]   // lancy
        [210].0   // PMP ETANG EN DEF
        [210].1   // no flow pumping from etang
        [210].2   // FLOW TOO LOW Q1
        [210].3   // LEVEL PRETREATED TOO HIGH
        [210].4   // LEVEL LOW PRETREATED WATER WARNING
        [210].5   // LEVEL LOW PRETREATED WATER
        [210].6   // ANORMAL EMPTYING PRETREATED WATER TANK
        [210].7   // 2 pump pretreated tank out of order P3&P4
        [210].8   // no flow pumping from PRETREATED WATER TANK
        [210].9   // FLOW TOO LOW Q2
        [210].11   // recup water tank L1 too high
        [210].12   // PMP RECUP L1 OUT OF ORDER
        [210].13   // recup water tank L2 too high
        [210].14   // PMP RECUP L2 OUT OF ORDER
        [210].15   // recup water tank L3 too high
        [211].0   // PMP RECUP L3 OUT OF ORDER
        [211].1   // recup water tank L4 too high
        [211].2   // PMP RECUP L4 OUT OF ORDER
        [211].3   // LEVEL NAOH TOO HIGH
        [211].4   // ANORMAL LEVEL DECREASE naoh TANK
        [211].5   // LACK DETECTIE NAOH
        [211].6   // LEVEL H2SO4 TOO HIGH
        [211].7   // ANORMAL LEVEL DECREASE H2SO4 TANK
        [211].8   // LACK DETECTIE H2SO4
        [211].9   // defaut niveau vijver trop bas
        [211].11   // memo defaut vanne position eau ville
        [226].0   // DE PLC statdemande soudestation
        [226].1   // DE PLC statdemandearret soude stat
        [226].2   // de plc ligne STATfc vanne soudeouverte
        [226].4   // de plc stationfc vanne soudefermée
        [230]   // lancy
        [245]   // quantité souderestante station
        [246].3   // vers plc statouvrir vannesoude
        [246].4   // vers plc statapport soudestat finit
        [246].5   // vers plc statapport soudeoccupé
        [246].6   // vers plc statapport soudestat accordé
        [246].7   // VERS PLC STATSOUDE VERS L1
        [246].8   // VERS PLC STATSOUDE VERS L2
        [246].9   // VERS PLC L1SOUDE VERS STAT
        [246].10   // VERS PLC STATSOUDE VERS L4
        [246].11   // VERS PLC STATSOUDE VERS STAT
   N11 : DINT[150] := ([0] := 4, [1] := 800, [2] := 75, [3] := 71, [4] := 55, [5] := 57, [6] := 4, [7] := 4, [8] := 4, [9] := 14528, [10] := 49, [11] := 4, [12] := 45, [14] := 4, [17] := 4, [18] := 4, [19] := 4, [20] := 8192, [21] := 30, [22] := 5, [23] := 7, [24] := 137, [25] := 50, [28] := 5, [34] := 4, [35] := 4, [36] := 4, [37] := 4, [50] := 48, [51] := 7, [52] := 1, [80] := 75, [81] := 75, [100] := 6, [101] := 609, [103] := 336, [104] := 5, [106] := 45, [108] := 45, [109] := 45);
        [10]   // debit venturi
        [20]   // message vers Lancy
        [50]   // msg vers lancy debit venturi
        [51]   // vers lancy defaut niveau 1
        [52]   // vers lancy defaut niveau 2
        [53]   // reserver vers lancy
        [54]   // reserver vers lancy
        [55]   // reserver vers lancy
        [80]   // de relalarm
        [81]   // de relalarm
   N12 : DINT[230] := ([0] := 430, [7] := 410, [8] := 322, [12] := 16332, [14] := 90, [15] := 188, [16] := 877, [20] := 126, [21] := 350, [23] := 309, [25] := 455, [26] := 6149, [27] := 6376, [30] := 357, [32] := 78, [34] := 258, [36] := 39, [38] := 999, [40] := 80, [42] := 79, [44] := -500, [50] := 103, [62] := 252, [63] := 301, [64] := -25, [66] := 72, [68] := -25, [70] := 15, [74] := 200, [76] := 172, [78] := 45, [79] := 79, [88] := 84, [90] := 88, [91] := 75, [92] := 93, [93] := 75, [94] := 58, [96] := -25, [98] := -35, [102] := 49, [106] := 839, [108] := 831, [110] := 95, [111] := 80, [112] := -1250, [113] := 731, [116] := -308, [118] := -25, [120] := -37, [121] := 29136, [122] := 97, [124] := -490, [126] := -25, [128] := -25, [131] := 367, [132] := 303, [133] := 215, [134] := 170, [135] := 164,
        [136] := 247, [137] := 242, [138] := 152, [140] := -25, [141] := -25, [142] := -25, [143] := -30, [144] := -35, [145] := 48, [146] := -725, [147] := -25, [148] := 192, [149] := 2798, [154] := 192, [155] := 2865, [156] := 125, [157] := 1708, [158] := 192, [159] := 2878, [160] := -75, [163] := 4, [172] := 3310, [174] := 7, [179] := 20, [180] := 250633, [181] := 1638, [182] := 453, [187] := -375, [188] := 453, [189] := 2634, [193] := 1, [197] := 3, [198] := 2, [199] := 6, [200] := 6, [201] := 2, [202] := 3, [203] := 2, [204] := 332, [205] := 215, [206] := 170, [207] := 165, [208] := 297, [209] := 242, [210] := 166, [211] := 450, [212] := 301, [213] := 638, [215] := 26, [216] := -24, [217] := -30, [218] := 341, [219] := 1000, [220] := 397, [221] := -250);
        [14]   // 0
        [15]   // Q1_ISTT_OPTEL_ONTIJ1 Q1 optelling aantal pulsen waterteller
        [16]   // Q1_ISTT_OPTEL_ONTIJ2 Q1 optelling aantal pulsen waterteller ontijzer 2
        [17]   // Q1_ISTT_TOTAAL Q1 optelling aantal pulsen waterteller totaal
        [20]   // Q2_ISTT_OPTEL_VERZ1 Q2 optelling aantal pulsen waterteller verzacher 1
        [21]   // Q2_ISTT_OPTEL_VERZ2 Q2 optelling aantal pulsen waterteller verzacher 2
        [22]   // total stfa 31 osmose
        [23]   // total stfa 32 osmose
        [30]   // IST_COND3 Ist waarde analoog ingang conductiviteit 3
        [32]   // LEVEL RECUP L1
        [34]   // ISST_CON4
        [36]   // LEVEL TANK RECUP L2
        [38]   // iana38
        [40]   // LEVEL TANK RECUP L3
        [42]   // niveau cuve AZ
        [46]   // IST_DEBIET_Q3 Ist waarde debiet Q3
        [50]   // IST_COND5 Ist waarde analoog ingang conductiviteit 5
        [60]   // TURBIDITEIT LANCY
        [62]   // puisard ibt
        [64]   // niveau puisard ligne 4
        [66]   // niveau vijver
        [68]   // HARDHEID hardheid controle
        [70]   // CDRO1 conductiviteit controle 1
        [72]   // CDRO2 conductiviteit controle 2
        [74]   // CDRO3 conductiviteit controle 3
        [76]   // debit osmose 1 permeat
        [78]   // debit osmose 1 concentrat
        [80]   // debit osmose 2 permeat
        [82]   // debit osmose 2 concentrat
        [84]   // debit osmose 3 permeat
        [86]   // debit osmose 3 concentrat
        [88]   // lus1 r?ervoir ptéraitement
        [90]   // debit Q2 vers ligne de production
        [92]   // debit Q3 de ligne de production
        [94]   // ISTT_WAARDE_PH11 ph 1.1 eau sale retour ligne neutralisation
        [96]   // zout level
        [98]   // ph 1.2 eau sale retour ligne neutralisation
        [100]   // 'reserve semble defectueux
        [102]   // IST_PH2 ph 2 eau recyclé
        [104]   // conductivit?,cond 7
        [106]   // ANAL_ING_NIV_LUS_2 Analoogingang niveua lus 2 niveau acide H2SO4
        [108]   // ANAL_ING_NIV_LUS_3 Analoogingang niveua lus 3 niveau NAOH
        [110]   // niveau lus 4 eau clarifié
        [112]   // ANAL_ING_CON1 cond 1 conductivit?,eau recyclé
        [114]   // debit eau ville en m?/h
        [116]   // cond 2 conductivit?,global osmose
        [120]   // Q4
        [124]   // ISST_CON6 cond 6
        [130]   // F8M80 total d?it puits 2
        [131]   // total debit puit 3
        [132]   // average level landeniaan L1
        [133]   // average level kijtlaag k1
        [134]   // average level Quartair Q1
        [135]   // average level Landeniaan L2
        [136]   // average level kijtlaag k2
        [137]   // average level landeniaan L3
        [138]   // average level quartair Q2
        [140]   // LEVEL TANK RECUP L4
        [141]   // debit put 2
        [142]   // debit put 1
        [143]   // debit put 3
        [144]   // ph venturi
        [145]   // debit venturi
        [146]   // conductivite venturi
        [147]   // tEMPERATURE venturi
        [148]   // nbr min pnp pro1 marche aujourd hui
        [149]   // nbr min pnp pro1 marche hier
        [150]   // nbr min pnp pro2 marche aujourd hui
        [151]   // nbr min pnp pro2 marche hier
        [152]   // nbr min pnp pro3 marche aujourd hui
        [153]   // nbr min pnp pro1 marche hier
        [155]   // heure rotat pmp L1
        [156]   // heure rotat pmp L2
        [159]   // heure rotat pmp L3
        [160]   // dh <- bassin T?venturi
        [161]   // dh <- bassin
        [162]   // dh <- bassin
        [163]   // dh <- bassin
        [164]   // dh <- bassin
        [165]   // dh <- bassin
        [166]   // dh <- bassin
        [167]   // dh <- bassin
        [168]   // dh <- bassin
        [169]   // dh <- bassin
        [171]   // heure rotat pmp L4
        [172]   // total debit eau péraité hier
        [189]   // total eau de retour vers neutral
        [204]   // Landeniaan L1
        [205]   // Krijtlaag K1
        [206]   // Quartair Q1
        [207]   // Landeniaan L2
        [208]   // Krijtlaag K2
        [209]   // Landeniaan L3
        [210]   // Quartair Q2
        [214]   // % run/heure pmp put 2
        [215]   // % run/heure pmp put 3
        [216]   // average flow pmp put 2
        [217]   // average flow pmp put 3
        [218]   // pression vers ligne
   N12_110 : REAL := 94.65171;
   N12_14 : REAL := 89.939995;
   N12_219 : REAL := 1000.0;
   N12_220 : REAL := 397.4975;
   N12_221 : REAL := -250.01907;
   N12_38 : REAL := 999.4;
   N12_44 : REAL := -500.2;
   N13 : DINT[230] := ([8] := 5, [10] := 6000, [11] := 60, [16] := 1000, [18] := 1000, [20] := 250, [21] := 350, [22] := 350, [23] := 350, [25] := 1000, [30] := 2500, [34] := 2500, [38] := 2500, [46] := 500, [47] := 80, [52] := 75, [53] := 80, [54] := 75, [56] := 3600, [57] := 80, [62] := 7500, [63] := 300, [68] := 20, [70] := 205, [72] := 205, [74] := 205, [79] := 60, [80] := 30, [81] := 75, [82] := 85, [83] := 60, [84] := 95, [87] := 60, [94] := 53, [95] := 90, [96] := 10, [98] := 10, [103] := 40, [104] := 90, [109] := 30, [110] := 35, [111] := 45, [112] := 3500, [113] := 50, [116] := 1500, [122] := 100, [124] := 2500, [125] := 1, [126] := 3600, [129] := 55, [130] := 105, [131] := 52, [132] := 84, [134] := 10, [135] := 831, [137] := 10, [139] := 10, [140] := 839, [150] := 85, [151] := 55,
        [152] := 85, [153] := 55, [154] := 85, [155] := 55, [156] := 85, [157] := 60, [160] := 261, [161] := 162, [162] := 242, [163] := 170, [164] := 131, [165] := 206, [166] := 230);
        [9]   // SOLL_SNEL_PD1_2 sollwaarde snelheid PD1 2
        [10]   // SOLL_TIJD_PD1_2_UIT sollwaarde flip flop uit pd1 en pd2
        [11]   // SOLL_TIJD_PD1_2_AAN sollwaarde flip flop aan pd1 en pd2
        [15]   // SOLL_TOT1_STFA11 soll waarde q1 stfa1.1
        [16]   // SOLL_TOT1_STFA12 soll waarde q1 stfa1.2
        [30]   // SOLL_COND3 Soll waarde conductiviteit 3
        [31]   // SOLL_ALARM_COND3 Soll waarde alarm conductiviteit 3
        [40]   // SOLL_COND4 Soll waarde conductiviteit 4
        [41]   // SOLL_ALARM_COND4 Soll waarde alarm conductiviteit 4
        [50]   // SOLL_COND5 Soll waarde conductiviteit 5
        [51]   // SOLL_ALARM_COND5 Soll waarde alarm conductiviteit 5
        [52]   // SUPERVISION REFERENCE SPEED PM2
        [53]   // supervision REFERENCE SPEED PM4
        [54]   // SUPERVISION SPEED REFERENCE PM1
        [57]   // supervision REFERENCE SPEED PM3
        [60]   // SOLL_COND6 Soll waarde conductiviteit 6
        [61]   // SOLL_ALARM_COND6 Soll waarde alarm conductiviteit 6
        [94]   // SOLL_MIN_BAZE_PH11 SOLL_waarde minimum instelling van lage ph baze
        [95]   // SOLL_MAX_ZUUR_PH11 SOLL_waarde max instelling van hoge ph zuur
        [103]   // SOL_PH2_MIN
        [104]   // SOL_PH2_MAX
        [129]   // niveau remplissage pompe arreté eau de ville
        [130]   // AUX LVL INTERMEDIAIRE ALARME BAS
        [131]   // LVL LOW WARNING PREATREAED WATER
        [132]   // EMO LVL PRETREATED WATER TANK
        [133]   // DELTA LVL PREATREATED WATER
        [134]   // CHUTE MAXI EN POMPAGE LVL PRETREATED WATER TANK
        [135]   // MEMO LVL NAOH TANK
